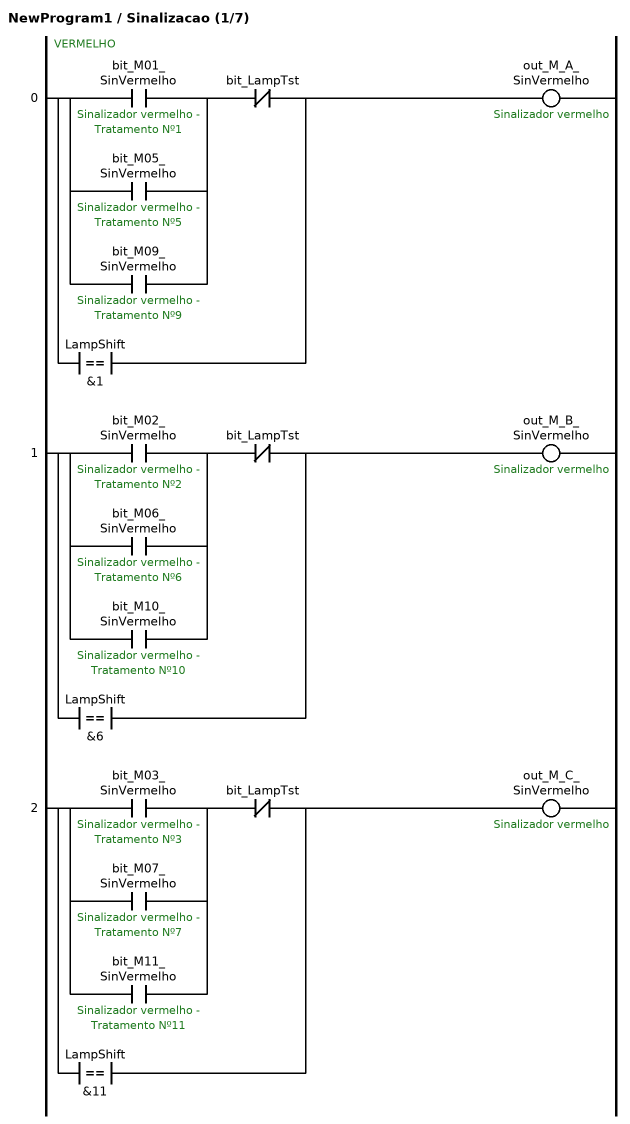
; [picture p48: NewProgram1 / Sinalizacao, rungs 0-2]
; rung 0: VERMELHO
LD bit_M01_SinVermelho  ; Sinalizador vermelho - Tratamento Nº1
OR bit_M05_SinVermelho  ; Sinalizador vermelho - Tratamento Nº5
OR bit_M09_SinVermelho  ; Sinalizador vermelho - Tratamento Nº9
ANDNOT bit_LampTst
OR=(300) LampShift &1
OUT out_M_A_SinVermelho  ; Sinalizador vermelho
; rung 1
LD bit_M02_SinVermelho  ; Sinalizador vermelho - Tratamento Nº2
OR bit_M06_SinVermelho  ; Sinalizador vermelho - Tratamento Nº6
OR bit_M10_SinVermelho  ; Sinalizador vermelho - Tratamento Nº10
ANDNOT bit_LampTst
OR=(300) LampShift &6
OUT out_M_B_SinVermelho  ; Sinalizador vermelho
; rung 2
LD bit_M03_SinVermelho  ; Sinalizador vermelho - Tratamento Nº3
OR bit_M07_SinVermelho  ; Sinalizador vermelho - Tratamento Nº7
OR bit_M11_SinVermelho  ; Sinalizador vermelho - Tratamento Nº11
ANDNOT bit_LampTst
OR=(300) LampShift &11
OUT out_M_C_SinVermelho  ; Sinalizador vermelho

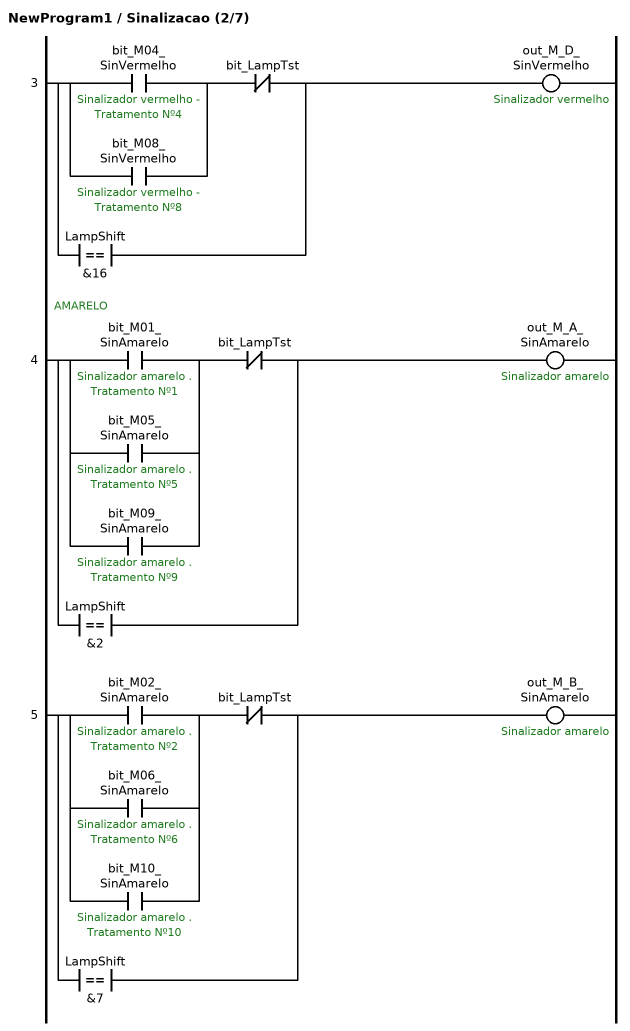
; rung 3
LD bit_M04_SinVermelho  ; Sinalizador vermelho - Tratamento Nº4
OR bit_M08_SinVermelho  ; Sinalizador vermelho - Tratamento Nº8
ANDNOT bit_LampTst
OR=(300) LampShift &16
OUT out_M_D_SinVermelho  ; Sinalizador vermelho
; rung 4: AMARELO
LD bit_M01_SinAmarelo  ; Sinalizador amarelo . Tratamento Nº1
OR bit_M05_SinAmarelo  ; Sinalizador amarelo . Tratamento Nº5
OR bit_M09_SinAmarelo  ; Sinalizador amarelo . Tratamento Nº9
ANDNOT bit_LampTst
OR=(300) LampShift &2
OUT out_M_A_SinAmarelo  ; Sinalizador amarelo
; rung 5
LD bit_M02_SinAmarelo  ; Sinalizador amarelo . Tratamento Nº2
OR bit_M06_SinAmarelo  ; Sinalizador amarelo . Tratamento Nº6
OR bit_M10_SinAmarelo  ; Sinalizador amarelo . Tratamento Nº10
ANDNOT bit_LampTst
OR=(300) LampShift &7
OUT out_M_B_SinAmarelo  ; Sinalizador amarelo

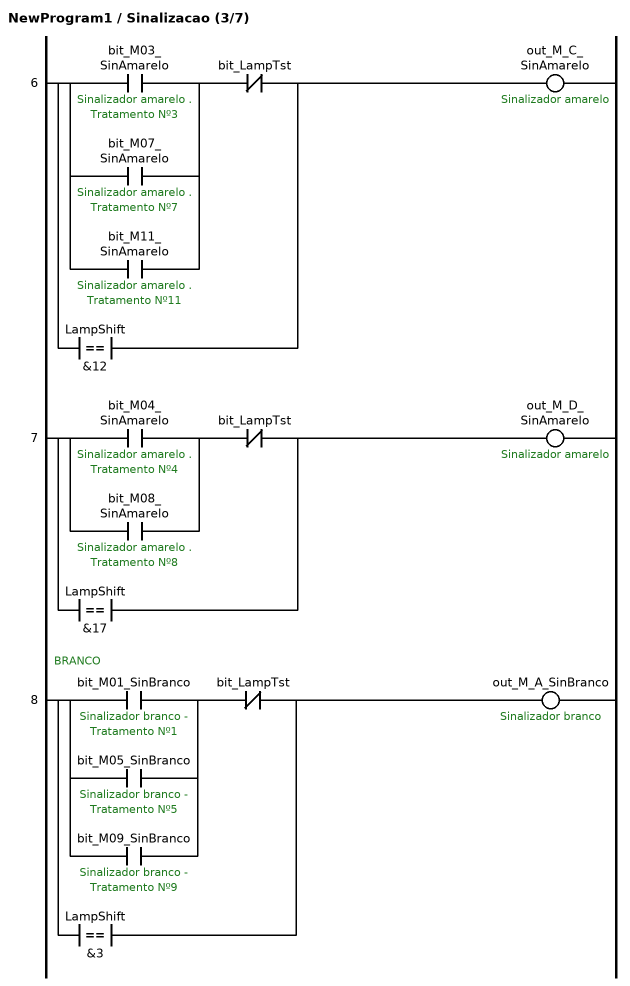
; rung 6
LD bit_M03_SinAmarelo  ; Sinalizador amarelo . Tratamento Nº3
OR bit_M07_SinAmarelo  ; Sinalizador amarelo . Tratamento Nº7
OR bit_M11_SinAmarelo  ; Sinalizador amarelo . Tratamento Nº11
ANDNOT bit_LampTst
OR=(300) LampShift &12
OUT out_M_C_SinAmarelo  ; Sinalizador amarelo
; rung 7
LD bit_M04_SinAmarelo  ; Sinalizador amarelo . Tratamento Nº4
OR bit_M08_SinAmarelo  ; Sinalizador amarelo . Tratamento Nº8
ANDNOT bit_LampTst
OR=(300) LampShift &17
OUT out_M_D_SinAmarelo  ; Sinalizador amarelo
; rung 8: BRANCO
LD bit_M01_SinBranco  ; Sinalizador branco - Tratamento Nº1
OR bit_M05_SinBranco  ; Sinalizador branco - Tratamento Nº5
OR bit_M09_SinBranco  ; Sinalizador branco - Tratamento Nº9
ANDNOT bit_LampTst
OR=(300) LampShift &3
OUT out_M_A_SinBranco  ; Sinalizador branco

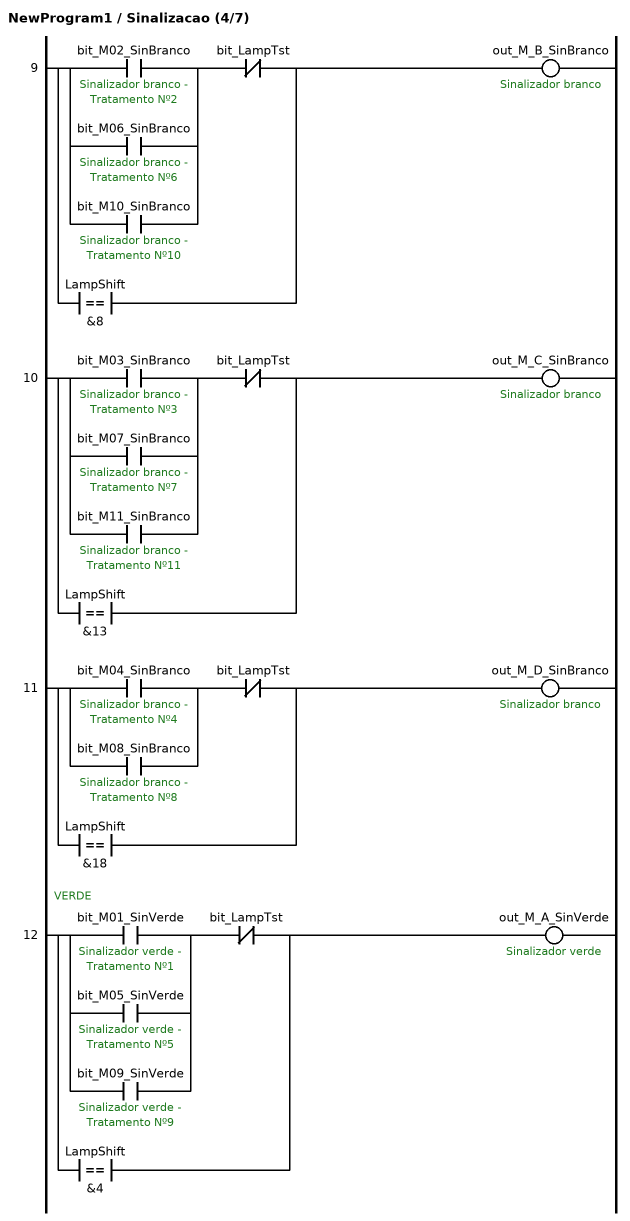
; rung 9
LD bit_M02_SinBranco  ; Sinalizador branco - Tratamento Nº2
OR bit_M06_SinBranco  ; Sinalizador branco - Tratamento Nº6
OR bit_M10_SinBranco  ; Sinalizador branco - Tratamento Nº10
ANDNOT bit_LampTst
OR=(300) LampShift &8
OUT out_M_B_SinBranco  ; Sinalizador branco
; rung 10
LD bit_M03_SinBranco  ; Sinalizador branco - Tratamento Nº3
OR bit_M07_SinBranco  ; Sinalizador branco - Tratamento Nº7
OR bit_M11_SinBranco  ; Sinalizador branco - Tratamento Nº11
ANDNOT bit_LampTst
OR=(300) LampShift &13
OUT out_M_C_SinBranco  ; Sinalizador branco
; rung 11
LD bit_M04_SinBranco  ; Sinalizador branco - Tratamento Nº4
OR bit_M08_SinBranco  ; Sinalizador branco - Tratamento Nº8
ANDNOT bit_LampTst
OR=(300) LampShift &18
OUT out_M_D_SinBranco  ; Sinalizador branco
; rung 12: VERDE
LD bit_M01_SinVerde  ; Sinalizador verde - Tratamento Nº1
OR bit_M05_SinVerde  ; Sinalizador verde - Tratamento Nº5
OR bit_M09_SinVerde  ; Sinalizador verde - Tratamento Nº9
ANDNOT bit_LampTst
OR=(300) LampShift &4
OUT out_M_A_SinVerde  ; Sinalizador verde

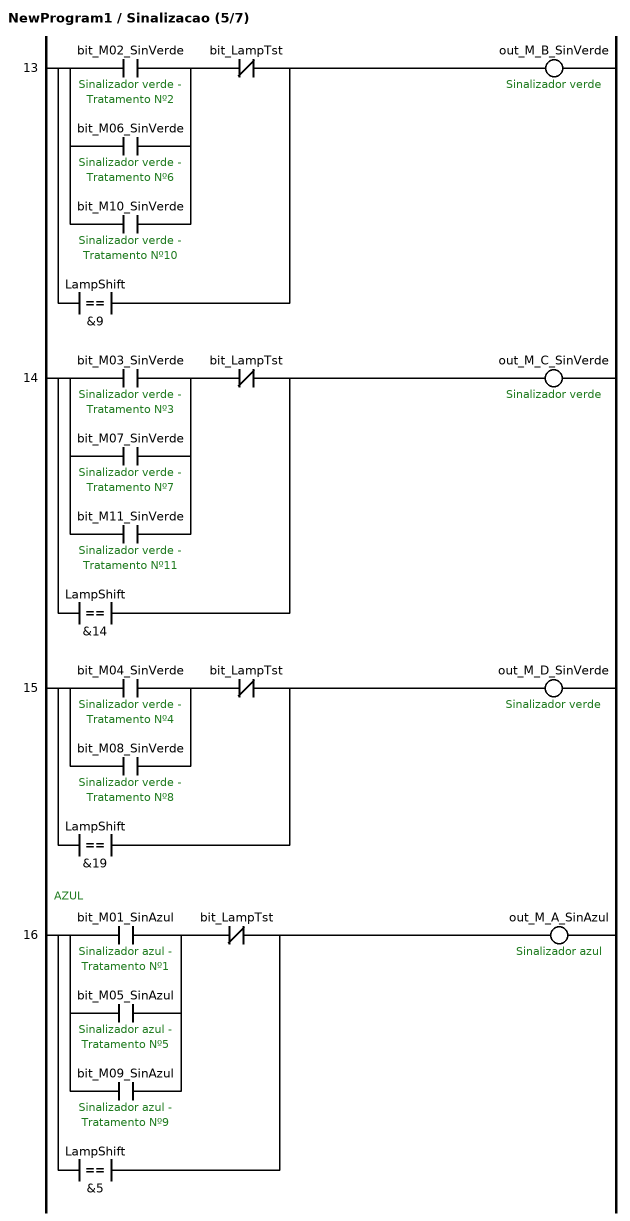
; rung 13
LD bit_M02_SinVerde  ; Sinalizador verde - Tratamento Nº2
OR bit_M06_SinVerde  ; Sinalizador verde - Tratamento Nº6
OR bit_M10_SinVerde  ; Sinalizador verde - Tratamento Nº10
ANDNOT bit_LampTst
OR=(300) LampShift &9
OUT out_M_B_SinVerde  ; Sinalizador verde
; rung 14
LD bit_M03_SinVerde  ; Sinalizador verde - Tratamento Nº3
OR bit_M07_SinVerde  ; Sinalizador verde - Tratamento Nº7
OR bit_M11_SinVerde  ; Sinalizador verde - Tratamento Nº11
ANDNOT bit_LampTst
OR=(300) LampShift &14
OUT out_M_C_SinVerde  ; Sinalizador verde
; rung 15
LD bit_M04_SinVerde  ; Sinalizador verde - Tratamento Nº4
OR bit_M08_SinVerde  ; Sinalizador verde - Tratamento Nº8
ANDNOT bit_LampTst
OR=(300) LampShift &19
OUT out_M_D_SinVerde  ; Sinalizador verde
; rung 16: AZUL
LD bit_M01_SinAzul  ; Sinalizador azul - Tratamento Nº1
OR bit_M05_SinAzul  ; Sinalizador azul - Tratamento Nº5
OR bit_M09_SinAzul  ; Sinalizador azul - Tratamento Nº9
ANDNOT bit_LampTst
OR=(300) LampShift &5
OUT out_M_A_SinAzul  ; Sinalizador azul

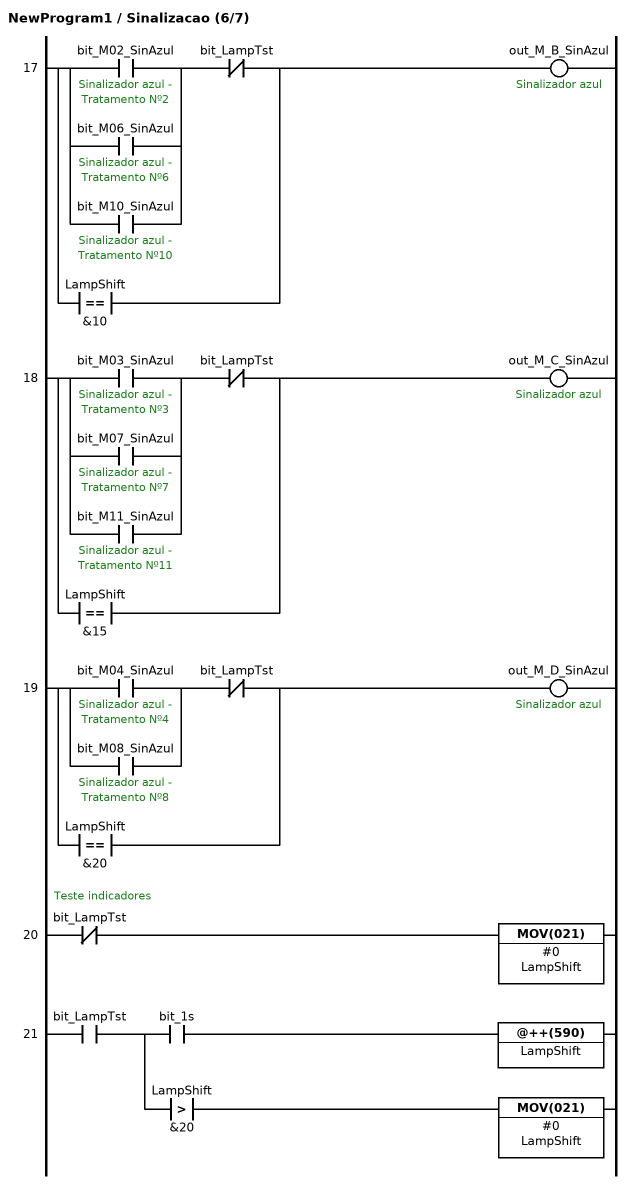
; rung 17
LD bit_M02_SinAzul  ; Sinalizador azul - Tratamento Nº2
OR bit_M06_SinAzul  ; Sinalizador azul - Tratamento Nº6
OR bit_M10_SinAzul  ; Sinalizador azul - Tratamento Nº10
ANDNOT bit_LampTst
OR=(300) LampShift &10
OUT out_M_B_SinAzul  ; Sinalizador azul
; rung 18
LD bit_M03_SinAzul  ; Sinalizador azul - Tratamento Nº3
OR bit_M07_SinAzul  ; Sinalizador azul - Tratamento Nº7
OR bit_M11_SinAzul  ; Sinalizador azul - Tratamento Nº11
ANDNOT bit_LampTst
OR=(300) LampShift &15
OUT out_M_C_SinAzul  ; Sinalizador azul
; rung 19
LD bit_M04_SinAzul  ; Sinalizador azul - Tratamento Nº4
OR bit_M08_SinAzul  ; Sinalizador azul - Tratamento Nº8
ANDNOT bit_LampTst
OR=(300) LampShift &20
OUT out_M_D_SinAzul  ; Sinalizador azul
; rung 20: Teste indicadores
LDNOT bit_LampTst
MOV(021) #0 LampShift
; rung 21
LD bit_LampTst
OUT TR0
AND bit_1s
@++(590) LampShift
LD TR0
AND>(320) LampShift &20
MOV(021) #0 LampShift

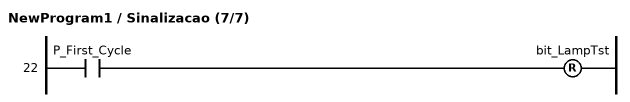
; rung 22
LD P_First_Cycle
RSET bit_LampTst

### Section RqstForTransfer

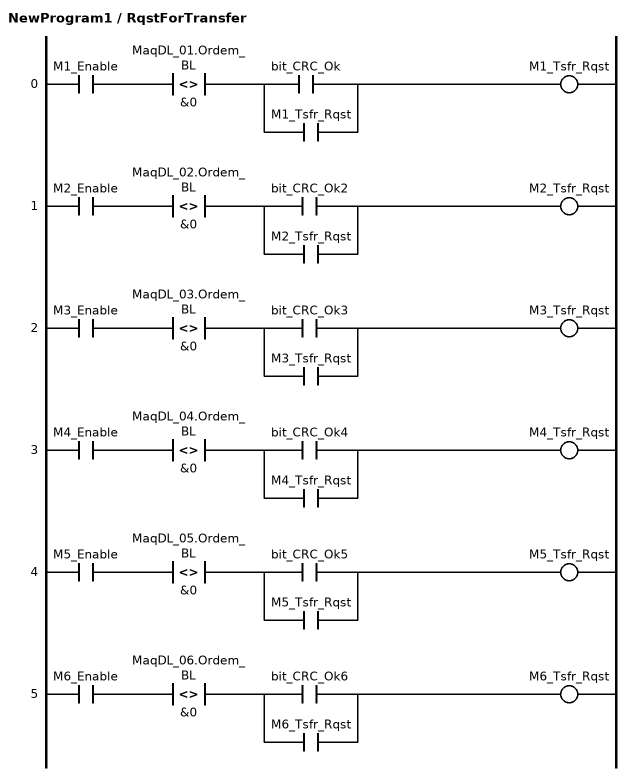
; rung 0
LD M1_Enable
AND<>(305) MaqDL_01.Ordem_BL &0
LD bit_CRC_Ok
OR M1_Tsfr_Rqst
ANDLD
OUT M1_Tsfr_Rqst
; rung 1
LD M2_Enable
AND<>(305) MaqDL_02.Ordem_BL &0
LD bit_CRC_Ok2
OR M2_Tsfr_Rqst
ANDLD
OUT M2_Tsfr_Rqst
; rung 2
LD M3_Enable
AND<>(305) MaqDL_03.Ordem_BL &0
LD bit_CRC_Ok3
OR M3_Tsfr_Rqst
ANDLD
OUT M3_Tsfr_Rqst
; rung 3
LD M4_Enable
AND<>(305) MaqDL_04.Ordem_BL &0
LD bit_CRC_Ok4
OR M4_Tsfr_Rqst
ANDLD
OUT M4_Tsfr_Rqst
; rung 4
LD M5_Enable
AND<>(305) MaqDL_05.Ordem_BL &0
LD bit_CRC_Ok5
OR M5_Tsfr_Rqst
ANDLD
OUT M5_Tsfr_Rqst
; rung 5
LD M6_Enable
AND<>(305) MaqDL_06.Ordem_BL &0
LD bit_CRC_Ok6
OR M6_Tsfr_Rqst
ANDLD
OUT M6_Tsfr_Rqst

### Section END

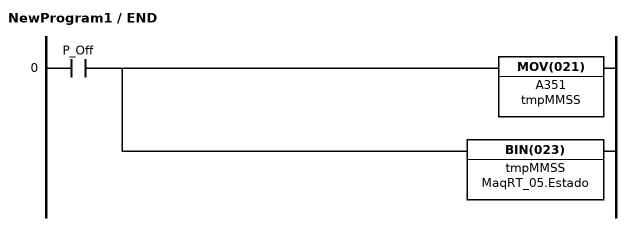
; rung 0
LD P_Off
MOV(021) A351 tmpMMSS
BIN(023) tmpMMSS MaqRT_05.Estado
; rung 1
END(001)

## Function block _CPU010_SendData (Omron library block, body left out)

## Function block ARRAY_COPY
VAR_INPUT
  NPos : INT;
END_VAR
VAR_IN_OUT
  ArIN : ARRAY[0..0] OF WORD;
  ArOUT : ARRAY[0..49] OF WORD;
END_VAR
VAR
  i : INT;
END_VAR
FOR i:= 0 TO 49 DO 
	ArOUT [i]:= 0;
END_FOR; 
FOR i:= 0 TO (NPos -1) DO 
	ArOUT [i]:= ArIN [i];
END_FOR; 

## Function block CopyRcp
VAR_INPUT
  Start : BOOL;
END_VAR
VAR_IN_OUT
  Dados : MqDL;
END_VAR
IF Start THEN
Dados.Cliente[0]:= Dados.Cliente_BL[0];
Dados.Cliente[1]:= Dados.Cliente_BL[1];
Dados.Cliente[2]:= Dados.Cliente_BL[2];
Dados.Cliente[3]:= Dados.Cliente_BL[3];
Dados.Cliente[4]:= Dados.Cliente_BL[4];
Dados.Cliente[5]:= Dados.Cliente_BL[5];
Dados.Cliente[6]:= Dados.Cliente_BL[6];
Dados.Cliente[7]:= Dados.Cliente_BL[7];
Dados.Cliente[8]:= Dados.Cliente_BL[8];
Dados.Cliente[9]:= Dados.Cliente_BL[9];
Dados.Cliente[10]:= Dados.Cliente_BL[10];
Dados.Cliente[11]:= Dados.Cliente_BL[11];
Dados.Cliente[12]:= Dados.Cliente_BL[12];
Dados.Cliente[13]:= Dados.Cliente_BL[13];
Dados.Cliente[14]:= Dados.Cliente_BL[14];
Dados.Cliente[15]:= Dados.Cliente_BL[15];
Dados.Cliente[16]:= Dados.Cliente_BL[16];
Dados.Cliente[17]:= Dados.Cliente_BL[17];
Dados.Cliente[18]:= Dados.Cliente_BL[18];
Dados.Cliente[19]:= Dados.Cliente_BL[19];
Dados.Cliente[20]:= Dados.Cliente_BL[20];
Dados.Cliente[21]:= Dados.Cliente_BL[21];
Dados.Cliente[22]:= Dados.Cliente_BL[22];
Dados.Cliente[23]:= Dados.Cliente_BL[23];
Dados.Cliente[24]:= Dados.Cliente_BL[24];
Dados.Cliente[25]:= Dados.Cliente_BL[25];
Dados.Cliente[26]:= Dados.Cliente_BL[26];
Dados.Cliente[27]:= Dados.Cliente_BL[27];
Dados.Cliente[28]:= Dados.Cliente_BL[28];
Dados.Cliente[29]:= Dados.Cliente_BL[29];
Dados.Cliente[30]:= Dados.Cliente_BL[30];
Dados.Cliente[31]:= Dados.Cliente_BL[31];
Dados.Cliente[32]:= Dados.Cliente_BL[32];
Dados.Cliente[33]:= Dados.Cliente_BL[33];
Dados.Cliente[34]:= Dados.Cliente_BL[34];
Dados.Cliente[35]:= Dados.Cliente_BL[35];
Dados.Cliente[36]:= Dados.Cliente_BL[36];
Dados.Cliente[37]:= Dados.Cliente_BL[37];
Dados.Cliente[38]:= Dados.Cliente_BL[38];
Dados.Cliente[39]:= Dados.Cliente_BL[39];
Dados.Cliente[40]:= Dados.Cliente_BL[40];
Dados.Cliente[41]:= Dados.Cliente_BL[41];
Dados.Cliente[42]:= Dados.Cliente_BL[42];
Dados.Cliente[43]:= Dados.Cliente_BL[43];
Dados.Cliente[44]:= Dados.Cliente_BL[44];
Dados.Cliente[45]:= Dados.Cliente_BL[45];
Dados.Cliente[46]:= Dados.Cliente_BL[46];
Dados.Cliente[47]:= Dados.Cliente_BL[47];
Dados.Cliente[48]:= Dados.Cliente_BL[48];
Dados.Cliente[49]:= Dados.Cliente_BL[49];

Dados.Artigo[0]:= Dados.Artigo_BL[0];
Dados.Artigo[1]:= Dados.Artigo_BL[1];
Dados.Artigo[2]:= Dados.Artigo_BL[2];
Dados.Artigo[3]:= Dados.Artigo_BL[3];
Dados.Artigo[4]:= Dados.Artigo_BL[4];
Dados.Artigo[5]:= Dados.Artigo_BL[5];
Dados.Artigo[6]:= Dados.Artigo_BL[6];
Dados.Artigo[7]:= Dados.Artigo_BL[7];
Dados.Artigo[8]:= Dados.Artigo_BL[8];
Dados.Artigo[9]:= Dados.Artigo_BL[9];
Dados.Artigo[10]:= Dados.Artigo_BL[10];
Dados.Artigo[11]:= Dados.Artigo_BL[11];
Dados.Artigo[12]:= Dados.Artigo_BL[12];
Dados.Artigo[13]:= Dados.Artigo_BL[13];
Dados.Artigo[14]:= Dados.Artigo_BL[14];
Dados.Artigo[15]:= Dados.Artigo_BL[15];
Dados.Artigo[16]:= Dados.Artigo_BL[16];
Dados.Artigo[17]:= Dados.Artigo_BL[17];
Dados.Artigo[18]:= Dados.Artigo_BL[18];
Dados.Artigo[19]:= Dados.Artigo_BL[19];
Dados.Artigo[20]:= Dados.Artigo_BL[20];
Dados.Artigo[21]:= Dados.Artigo_BL[21];
Dados.Artigo[22]:= Dados.Artigo_BL[22];
Dados.Artigo[23]:= Dados.Artigo_BL[23];
Dados.Artigo[24]:= Dados.Artigo_BL[24];
Dados.Artigo[25]:= Dados.Artigo_BL[25];
Dados.Artigo[26]:= Dados.Artigo_BL[26];
Dados.Artigo[27]:= Dados.Artigo_BL[27];
Dados.Artigo[28]:= Dados.Artigo_BL[28];
Dados.Artigo[29]:= Dados.Artigo_BL[29];
Dados.Artigo[30]:= Dados.Artigo_BL[30];
Dados.Artigo[31]:= Dados.Artigo_BL[31];
Dados.Artigo[32]:= Dados.Artigo_BL[32];
Dados.Artigo[33]:= Dados.Artigo_BL[33];
Dados.Artigo[34]:= Dados.Artigo_BL[34];
Dados.Artigo[35]:= Dados.Artigo_BL[35];
Dados.Artigo[36]:= Dados.Artigo_BL[36];
Dados.Artigo[37]:= Dados.Artigo_BL[37];
Dados.Artigo[38]:= Dados.Artigo_BL[38];
Dados.Artigo[39]:= Dados.Artigo_BL[39];
Dados.Artigo[40]:= Dados.Artigo_BL[40];
Dados.Artigo[41]:= Dados.Artigo_BL[41];
Dados.Artigo[42]:= Dados.Artigo_BL[42];
Dados.Artigo[43]:= Dados.Artigo_BL[43];
Dados.Artigo[44]:= Dados.Artigo_BL[44];
Dados.Artigo[45]:= Dados.Artigo_BL[45];
Dados.Artigo[46]:= Dados.Artigo_BL[46];
Dados.Artigo[47]:= Dados.Artigo_BL[47];
Dados.Artigo[48]:= Dados.Artigo_BL[48];
Dados.Artigo[49]:= Dados.Artigo_BL[49];

Dados.Encomenda[0]:= Dados.Encomenda_BL[0];
Dados.Encomenda[1]:= Dados.Encomenda_BL[1];
Dados.Encomenda[2]:= Dados.Encomenda_BL[2];
Dados.Encomenda[3]:= Dados.Encomenda_BL[3];
Dados.Encomenda[4]:= Dados.Encomenda_BL[4];
Dados.Encomenda[5]:= Dados.Encomenda_BL[5];
Dados.Encomenda[6]:= Dados.Encomenda_BL[6];
Dados.Encomenda[7]:= Dados.Encomenda_BL[7];
Dados.Encomenda[8]:= Dados.Encomenda_BL[8];
Dados.Encomenda[9]:= Dados.Encomenda_BL[9];
Dados.Encomenda[10]:= Dados.Encomenda_BL[10];
Dados.Encomenda[11]:= Dados.Encomenda_BL[11];
Dados.Encomenda[12]:= Dados.Encomenda_BL[12];
Dados.Encomenda[13]:= Dados.Encomenda_BL[13];
Dados.Encomenda[14]:= Dados.Encomenda_BL[14];
Dados.Encomenda[15]:= Dados.Encomenda_BL[15];
Dados.Encomenda[16]:= Dados.Encomenda_BL[16];
Dados.Encomenda[17]:= Dados.Encomenda_BL[17];
Dados.Encomenda[18]:= Dados.Encomenda_BL[18];
Dados.Encomenda[19]:= Dados.Encomenda_BL[19];
Dados.Encomenda[20]:= Dados.Encomenda_BL[20];
Dados.Encomenda[21]:= Dados.Encomenda_BL[21];
Dados.Encomenda[22]:= Dados.Encomenda_BL[22];
Dados.Encomenda[23]:= Dados.Encomenda_BL[23];
Dados.Encomenda[24]:= Dados.Encomenda_BL[24];
Dados.Encomenda[25]:= Dados.Encomenda_BL[25];
Dados.Encomenda[26]:= Dados.Encomenda_BL[26];
Dados.Encomenda[27]:= Dados.Encomenda_BL[27];
Dados.Encomenda[28]:= Dados.Encomenda_BL[28];
Dados.Encomenda[29]:= Dados.Encomenda_BL[29];
Dados.Encomenda[30]:= Dados.Encomenda_BL[30];
Dados.Encomenda[31]:= Dados.Encomenda_BL[31];
Dados.Encomenda[32]:= Dados.Encomenda_BL[32];
Dados.Encomenda[33]:= Dados.Encomenda_BL[33];
Dados.Encomenda[34]:= Dados.Encomenda_BL[34];
Dados.Encomenda[35]:= Dados.Encomenda_BL[35];
Dados.Encomenda[36]:= Dados.Encomenda_BL[36];
Dados.Encomenda[37]:= Dados.Encomenda_BL[37];
Dados.Encomenda[38]:= Dados.Encomenda_BL[38];
Dados.Encomenda[39]:= Dados.Encomenda_BL[39];
Dados.Encomenda[40]:= Dados.Encomenda_BL[40];
Dados.Encomenda[41]:= Dados.Encomenda_BL[41];
Dados.Encomenda[42]:= Dados.Encomenda_BL[42];
Dados.Encomenda[43]:= Dados.Encomenda_BL[43];
Dados.Encomenda[44]:= Dados.Encomenda_BL[44];
Dados.Encomenda[45]:= Dados.Encomenda_BL[45];
Dados.Encomenda[46]:= Dados.Encomenda_BL[46];
Dados.Encomenda[47]:= Dados.Encomenda_BL[47];
Dados.Encomenda[48]:= Dados.Encomenda_BL[48];
Dados.Encomenda[49]:= Dados.Encomenda_BL[49];

Dados.NomeReceita[0]:= Dados.NomeReceita_BL[0];
Dados.NomeReceita[1]:= Dados.NomeReceita_BL[1];
Dados.NomeReceita[2]:= Dados.NomeReceita_BL[2];
Dados.NomeReceita[3]:= Dados.NomeReceita_BL[3];
Dados.NomeReceita[4]:= Dados.NomeReceita_BL[4];
Dados.NomeReceita[5]:= Dados.NomeReceita_BL[5];
Dados.NomeReceita[6]:= Dados.NomeReceita_BL[6];
Dados.NomeReceita[7]:= Dados.NomeReceita_BL[7];
Dados.NomeReceita[8]:= Dados.NomeReceita_BL[8];
Dados.NomeReceita[9]:= Dados.NomeReceita_BL[9];
Dados.NomeReceita[10]:= Dados.NomeReceita_BL[10];
Dados.NomeReceita[11]:= Dados.NomeReceita_BL[11];
Dados.NomeReceita[12]:= Dados.NomeReceita_BL[12];
Dados.NomeReceita[13]:= Dados.NomeReceita_BL[13];
Dados.NomeReceita[14]:= Dados.NomeReceita_BL[14];
Dados.NomeReceita[15]:= Dados.NomeReceita_BL[15];
Dados.NomeReceita[16]:= Dados.NomeReceita_BL[16];
Dados.NomeReceita[17]:= Dados.NomeReceita_BL[17];
Dados.NomeReceita[18]:= Dados.NomeReceita_BL[18];
Dados.NomeReceita[19]:= Dados.NomeReceita_BL[19];
Dados.NomeReceita[20]:= Dados.NomeReceita_BL[20];
Dados.NomeReceita[21]:= Dados.NomeReceita_BL[21];
Dados.NomeReceita[22]:= Dados.NomeReceita_BL[22];
Dados.NomeReceita[23]:= Dados.NomeReceita_BL[23];
Dados.NomeReceita[24]:= Dados.NomeReceita_BL[24];
Dados.NomeReceita[25]:= Dados.NomeReceita_BL[25];
Dados.NomeReceita[26]:= Dados.NomeReceita_BL[26];
Dados.NomeReceita[27]:= Dados.NomeReceita_BL[27];
Dados.NomeReceita[28]:= Dados.NomeReceita_BL[28];
Dados.NomeReceita[29]:= Dados.NomeReceita_BL[29];
Dados.NomeReceita[30]:= Dados.NomeReceita_BL[30];
Dados.NomeReceita[31]:= Dados.NomeReceita_BL[31];
Dados.NomeReceita[32]:= Dados.NomeReceita_BL[32];
Dados.NomeReceita[33]:= Dados.NomeReceita_BL[33];
Dados.NomeReceita[34]:= Dados.NomeReceita_BL[34];
Dados.NomeReceita[35]:= Dados.NomeReceita_BL[35];
Dados.NomeReceita[36]:= Dados.NomeReceita_BL[36];
Dados.NomeReceita[37]:= Dados.NomeReceita_BL[37];
Dados.NomeReceita[38]:= Dados.NomeReceita_BL[38];
Dados.NomeReceita[39]:= Dados.NomeReceita_BL[39];
Dados.NomeReceita[40]:= Dados.NomeReceita_BL[40];
Dados.NomeReceita[41]:= Dados.NomeReceita_BL[41];
Dados.NomeReceita[42]:= Dados.NomeReceita_BL[42];
Dados.NomeReceita[43]:= Dados.NomeReceita_BL[43];
Dados.NomeReceita[44]:= Dados.NomeReceita_BL[44];
Dados.NomeReceita[45]:= Dados.NomeReceita_BL[45];
Dados.NomeReceita[46]:= Dados.NomeReceita_BL[46];
Dados.NomeReceita[47]:= Dados.NomeReceita_BL[47];
Dados.NomeReceita[48]:= Dados.NomeReceita_BL[48];
Dados.NomeReceita[49]:= Dados.NomeReceita_BL[49];

Dados.DataExpedic[0]:= Dados.DataExpedic_BL[0];
Dados.DataExpedic[1]:= Dados.DataExpedic_BL[1];
Dados.DataExpedic[2]:= Dados.DataExpedic_BL[2];
Dados.DataExpedic[3]:= Dados.DataExpedic_BL[3];

Dados.QtdEncom:= Dados.QtdEncom_BL;
Dados.QtdReal:= Dados.QtdReal_BL;

END_IF;

## Function block CopySteps
VAR_OUTPUT
  Rcp_Ok : BOOL;
END_VAR
VAR_IN_OUT
  Recipe : s_of;
  Steps : ARRAY[0..11] OF Passos;
END_VAR
Steps[0].f:= Recipe.prg.pss[0].f;
Steps[0].p1:= Recipe.prg.pss[0].p1;
Steps[0].p2:= Recipe.prg.pss[0].p2 ;

Steps[1].f:= Recipe.prg.pss[1].f;
Steps[1].p1:= Recipe.prg.pss[1].p1;
Steps[1].p2:= Recipe.prg.pss[1].p2 ;

Steps[2].f:= Recipe.prg.pss[2].f;
Steps[2].p1:= Recipe.prg.pss[2].p1;
Steps[2].p2:= Recipe.prg.pss[2].p2 ;

Steps[3].f:= Recipe.prg.pss[3].f;
Steps[3].p1:= Recipe.prg.pss[3].p1;
Steps[3].p2:= Recipe.prg.pss[3].p2 ;

Steps[4].f:= Recipe.prg.pss[4].f;
Steps[4].p1:= Recipe.prg.pss[4].p1;
Steps[4].p2:= Recipe.prg.pss[4].p2 ;

Steps[5].f:= Recipe.prg.pss[5].f;
Steps[5].p1:= Recipe.prg.pss[5].p1;
Steps[5].p2:= Recipe.prg.pss[5].p2 ;

Steps[6].f:= Recipe.prg.pss[6].f;
Steps[6].p1:= Recipe.prg.pss[6].p1;
Steps[6].p2:= Recipe.prg.pss[6].p2 ;

Steps[7].f:= Recipe.prg.pss[7].f;
Steps[7].p1:= Recipe.prg.pss[7].p1;
Steps[7].p2:= Recipe.prg.pss[7].p2 ;

Steps[8].f:= Recipe.prg.pss[8].f;
Steps[8].p1:= Recipe.prg.pss[8].p1;
Steps[8].p2:= Recipe.prg.pss[8].p2 ;

Steps[9].f:= Recipe.prg.pss[9].f;
Steps[9].p1:= Recipe.prg.pss[9].p1;
Steps[9].p2:= Recipe.prg.pss[9].p2 ;

Steps[10].f:= Recipe.prg.pss[10].f;
Steps[10].p1:= Recipe.prg.pss[10].p1;
Steps[10].p2:= Recipe.prg.pss[10].p2 ;

Steps[11].f:= Recipe.prg.pss[11].f;
Steps[11].p1:= Recipe.prg.pss[11].p1;
Steps[11].p2:= Recipe.prg.pss[11].p2 ;

Rcp_Ok:= TRUE;

## Function block CRC16
VAR_INPUT
  Bytes_Qty : INT;
  Swap : BOOL;  (* Swap LSB with MSB *)
  CRC_Ini : WORD;
END_VAR
VAR_OUTPUT
  CRC16 : WORD;
END_VAR
VAR_IN_OUT
  Str : STRING;
END_VAR
VAR
  Flip_Flop : BOOL;
  Next_Byte : WORD;
  CRC_Temp : WORD;
  i : INT;
  aux_Byte : WORD;
END_VAR

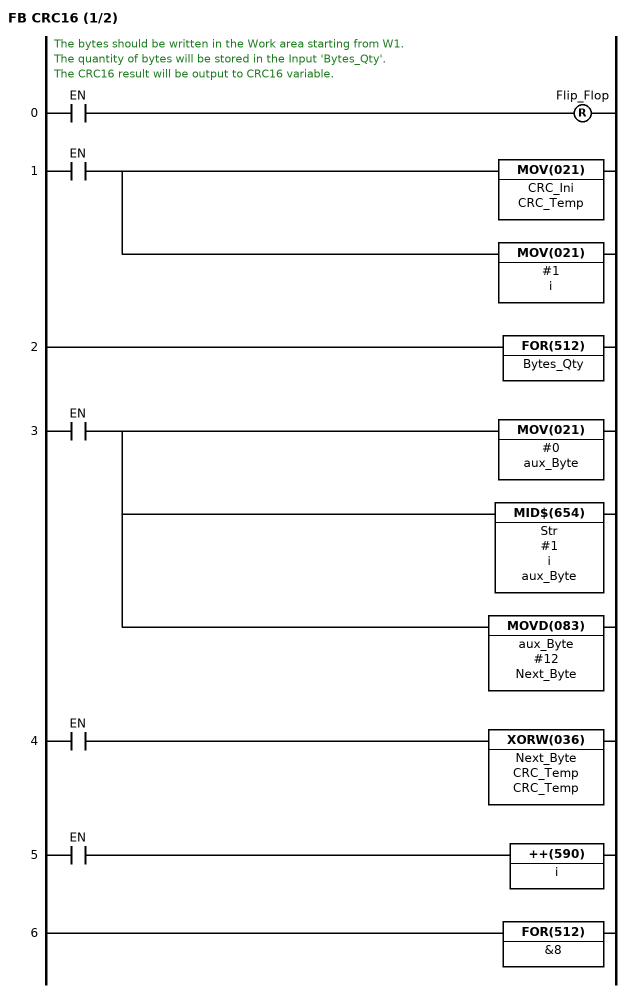
; rung 0: The bytes should be written in the Work area starting from W1. / The quantity of bytes will be stored in the Input 'Bytes_Qty'. / The CRC16 result will be output to CRC16 variable.
LD EN
RSET Flip_Flop
; rung 1
LD EN
MOV(021) CRC_Ini CRC_Temp
MOV(021) #1 i
; rung 2
FOR(512) Bytes_Qty
; rung 3
LD EN
MOV(021) #0 aux_Byte
MID$(654) Str #1 i aux_Byte
MOVD(083) aux_Byte #12 Next_Byte
; rung 4
LD EN
XORW(036) Next_Byte CRC_Temp CRC_Temp
; rung 5
LD EN
++(590) i
; rung 6
FOR(512) &8

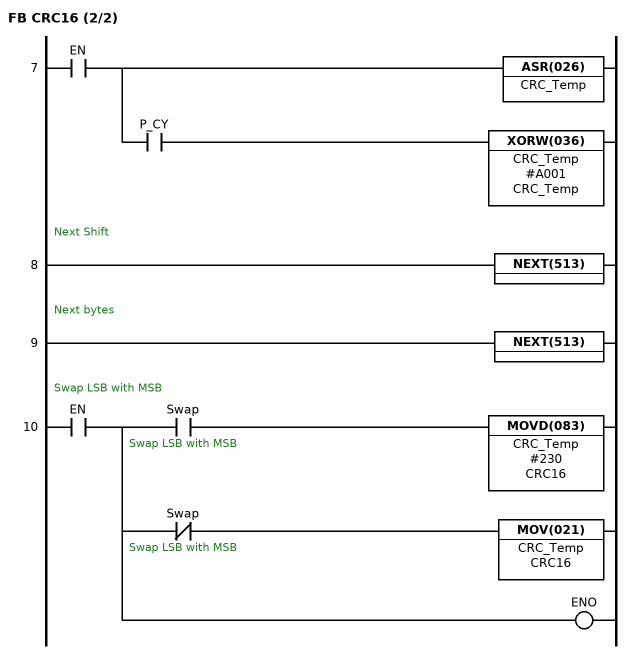
; rung 7
LD EN
ASR(026) CRC_Temp
AND P_CY
XORW(036) CRC_Temp #A001 CRC_Temp
; rung 8: Next Shift
NEXT(513)
; rung 9: Next bytes
NEXT(513)
; rung 10: Swap LSB with MSB
LD EN
OUT TR0
AND Swap  ; Swap LSB with MSB
MOVD(083) CRC_Temp #230 CRC16
LD TR0
ANDNOT Swap  ; Swap LSB with MSB
MOV(021) CRC_Temp CRC16
LD TR0
OUT ENO

## Function block DWord_To_Real
VAR_INPUT
  A : DWORD;
END_VAR
VAR_OUTPUT
  B : REAL;
END_VAR
VAR
  c : DINT;
END_VAR
c:= DWORD_TO_DINT(A);
B:= DINT_TO_REAL(c);

## Function block Empty_LSP
VAR_INPUT
  Fst_indx : INT;
  Lst_indx : INT;
END_VAR
VAR_OUTPUT
  Empty_Pos : INT;
  Last_Position : BOOL;
END_VAR
VAR_IN_OUT
  Ary : ARRAY[0..99] OF INT;
END_VAR
VAR
  itr : INT;
  Loop_Stop : BOOL;
END_VAR
Loop_Stop := FALSE;

FOR itr := Fst_indx TO Lst_indx DO
IF Ary[itr]=0 AND  NOT Loop_Stop THEN
	Empty_Pos := itr;
	Loop_Stop := TRUE;
END_IF;
END_FOR;

IF Ary[Lst_indx] <> 0 THEN
	Last_Position := TRUE;
	Empty_Pos := -1;
ELSE
	Last_Position := FALSE;
END_IF;

## Function block FIFO
; This function finds the least significant position of a arry. / The seeking area can be limited by firsr arry (FstAry) and last Array (LstAry) which are the inputs of function block.
VAR_INPUT
  Line_Free : BOOL;
  cmd_EN : BOOL;
  M1_Rqst : BOOL;
  M2_Rqst : BOOL;
  M3_Rqst : BOOL;
  M4_Rqst : BOOL;
  M5_Rqst : BOOL;
  M6_Rqst : BOOL;
  Table_Length : INT;
END_VAR
VAR_OUTPUT
  Actv_M : INT;
  cmd_M1 : BOOL;
  cmd_M2 : BOOL;
  cmd_M3 : BOOL;
  cmd_M4 : BOOL;
  cmd_M5 : BOOL;
  cmd_M6 : BOOL;
  Table_Full : BOOL;
END_VAR
VAR_IN_OUT
  Table : ARRAY[0..99] OF INT;
END_VAR
VAR
  M_Rqst_tmp : INT;
  Empty_in_Table : Empty_LSP;
  Empty_Position : INT;
  Shift_Table : Shift_Ary;
  cmd_Shift : BOOL;
  Tabel_LstIndx : INT;
END_VAR

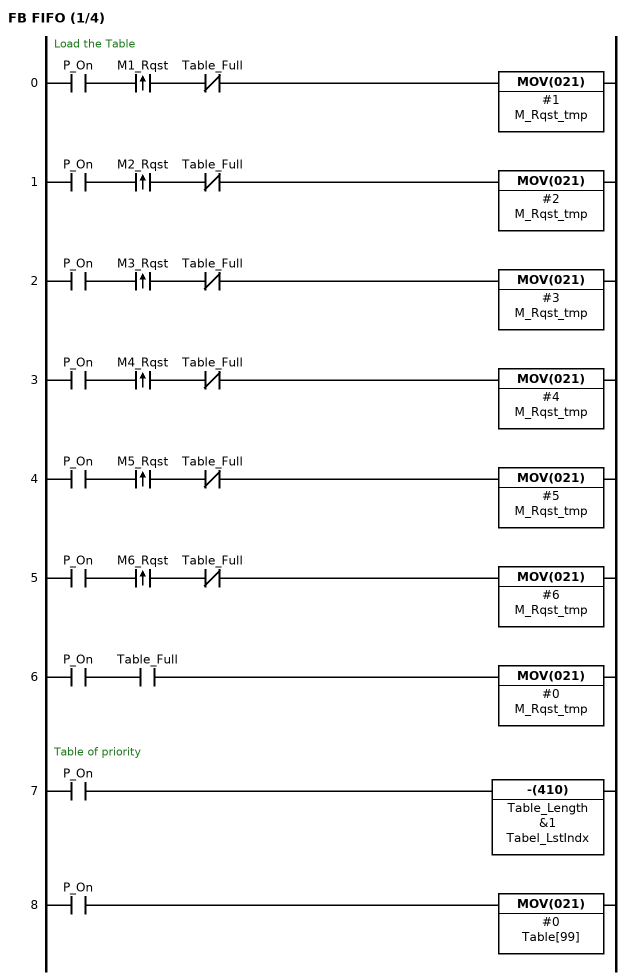
; rung 0: Load the Table
LD P_On
@AND M1_Rqst
ANDNOT Table_Full
MOV(021) #1 M_Rqst_tmp
; rung 1
LD P_On
@AND M2_Rqst
ANDNOT Table_Full
MOV(021) #2 M_Rqst_tmp
; rung 2
LD P_On
@AND M3_Rqst
ANDNOT Table_Full
MOV(021) #3 M_Rqst_tmp
; rung 3
LD P_On
@AND M4_Rqst
ANDNOT Table_Full
MOV(021) #4 M_Rqst_tmp
; rung 4
LD P_On
@AND M5_Rqst
ANDNOT Table_Full
MOV(021) #5 M_Rqst_tmp
; rung 5
LD P_On
@AND M6_Rqst
ANDNOT Table_Full
MOV(021) #6 M_Rqst_tmp
; rung 6
LD P_On
AND Table_Full
MOV(021) #0 M_Rqst_tmp
; rung 7: Table of priority
LD P_On
-(410) Table_Length &1 Tabel_LstIndx
; rung 8
LD P_On
MOV(021) #0 Table[99]

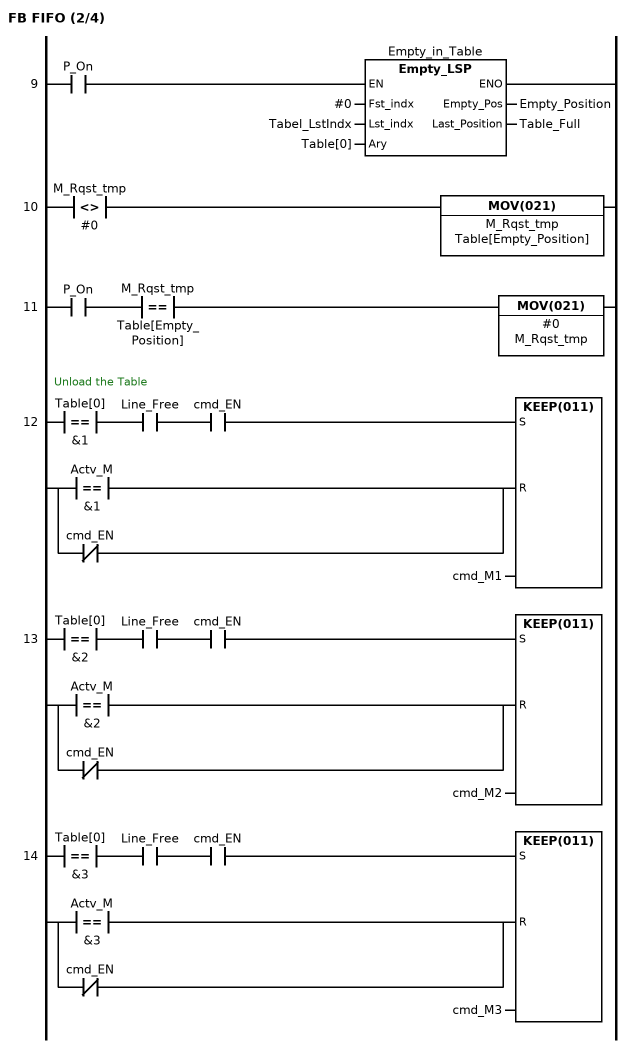
; rung 9
LD P_On
CALL Empty_in_Table : Empty_LSP (Fst_indx := #0, Lst_indx := Tabel_LstIndx, Ary := Table[0], Empty_Pos => Empty_Position, Last_Position => Table_Full)
; rung 10
LD<>(305) M_Rqst_tmp #0
MOV(021) M_Rqst_tmp Table[Empty_Position]
; rung 11
LD P_On
AND=(300) M_Rqst_tmp Table[Empty_Position]
MOV(021) #0 M_Rqst_tmp
; rung 12: Unload the Table
LD=(300) Table[0] &1
AND Line_Free
AND cmd_EN
LD=(300) Actv_M &1
ORNOT cmd_EN
KEEP(011) cmd_M1
; rung 13
LD=(300) Table[0] &2
AND Line_Free
AND cmd_EN
LD=(300) Actv_M &2
ORNOT cmd_EN
KEEP(011) cmd_M2
; rung 14
LD=(300) Table[0] &3
AND Line_Free
AND cmd_EN
LD=(300) Actv_M &3
ORNOT cmd_EN
KEEP(011) cmd_M3

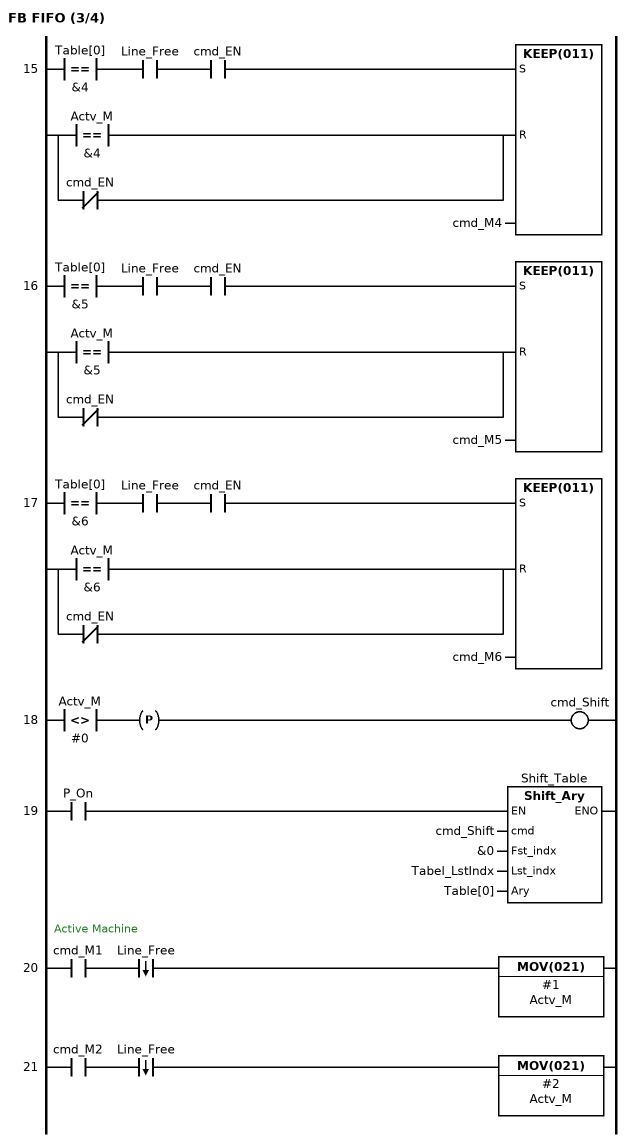
; rung 15
LD=(300) Table[0] &4
AND Line_Free
AND cmd_EN
LD=(300) Actv_M &4
ORNOT cmd_EN
KEEP(011) cmd_M4
; rung 16
LD=(300) Table[0] &5
AND Line_Free
AND cmd_EN
LD=(300) Actv_M &5
ORNOT cmd_EN
KEEP(011) cmd_M5
; rung 17
LD=(300) Table[0] &6
AND Line_Free
AND cmd_EN
LD=(300) Actv_M &6
ORNOT cmd_EN
KEEP(011) cmd_M6
; rung 18
LD<>(305) Actv_M #0
UP(521)
OUT cmd_Shift
; rung 19
LD P_On
CALL Shift_Table : Shift_Ary (cmd := cmd_Shift, Fst_indx := &0, Lst_indx := Tabel_LstIndx, Ary := Table[0])
; rung 20: Active Machine
LD cmd_M1
%AND Line_Free
MOV(021) #1 Actv_M
; rung 21
LD cmd_M2
%AND Line_Free
MOV(021) #2 Actv_M

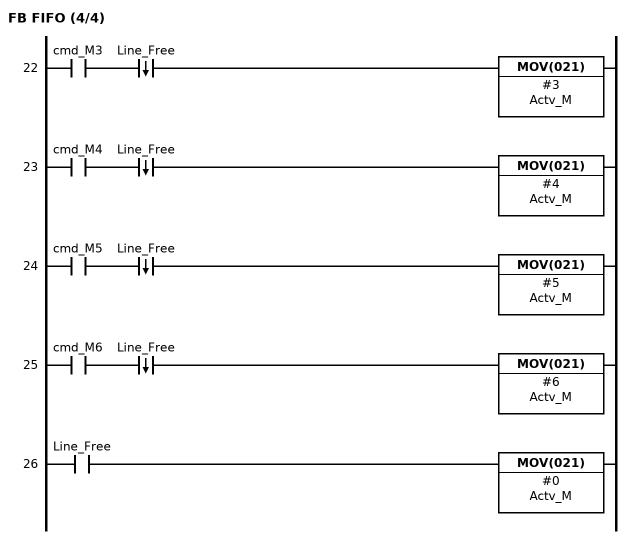
; rung 22
LD cmd_M3
%AND Line_Free
MOV(021) #3 Actv_M
; rung 23
LD cmd_M4
%AND Line_Free
MOV(021) #4 Actv_M
; rung 24
LD cmd_M5
%AND Line_Free
MOV(021) #5 Actv_M
; rung 25
LD cmd_M6
%AND Line_Free
MOV(021) #6 Actv_M
; rung 26
LD Line_Free
MOV(021) #0 Actv_M

## Function block PLC_to_MES
VAR_IN_OUT
  Dados : MqRT;
  BatchReal : s_Steps;
  Estado : s_Estado;
END_VAR
VAR
  Fnc : INT;
  P2_DInt : DINT;
  P1 : INT;
END_VAR
(* BATCH REAL *)
Fnc:= BatchReal.f;
P1:= BatchReal.p1;
P2_DInt:= REAL_TO_DINT(BatchReal.p2);

(*Limpa*)
Dados.BatchReal.Dedu.Active:= FALSE;
Dados.BatchReal.Heat.Active:= FALSE;
Dados.BatchReal.Inje.Active:= FALSE;
Dados.BatchReal.Load.Active:= FALSE;
Dados.BatchReal.Tumb.Active:= FALSE;
Dados.BatchReal.Unload.Active:= FALSE;
CASE Fnc OF 
	70: 
		Dados.BatchReal.Load.Active:= TRUE;
		Dados.BatchReal.Load.Value01:= INT_TO_DWORD(P1);
		Dados.BatchReal.Load.Value02:= DINT_TO_DWORD(P2_DInt);
	80:
		Dados.BatchReal.Unload.Active:= TRUE;
		Dados.BatchReal.Unload.Value01:= INT_TO_DWORD(P1);
		Dados.BatchReal.Unload.Value02:= DINT_TO_DWORD(P2_DInt);
	20:
		Dados.BatchReal.Heat.Active:= TRUE;
		Dados.BatchReal.Heat.Value01:= INT_TO_DWORD(P1);
		Dados.BatchReal.Heat.Value02:= DINT_TO_DWORD(P2_DInt);
	10:
		Dados.BatchReal.Dedu.Active:= TRUE;
		Dados.BatchReal.Dedu.Value01:= INT_TO_DWORD(P1);
		Dados.BatchReal.Dedu.Value02:= DINT_TO_DWORD(P2_DInt);
	40:
		Dados.BatchReal.Inje.Active:= TRUE;
		Dados.BatchReal.Inje.Value01:= INT_TO_DWORD(P1);
		Dados.BatchReal.Inje.Value02:= DINT_TO_DWORD(P2_DInt);
	30:
		Dados.BatchReal.Tumb.Active:= TRUE;
		Dados.BatchReal.Tumb.Value01:= INT_TO_DWORD(P1);
		Dados.BatchReal.Tumb.Value02:= DINT_TO_DWORD(P2_DInt);
END_CASE; 

(*ESTADOS*)
Dados.Ciclo:= Estado.Ciclo;
IF Estado.Estado AND NOT Estado.Avaria THEN
	Dados.Estado:= 1;	
ELSE
	Dados.Estado:= 0;
END_IF;
IF Estado.Manual THEN
	Dados.Estado:= 2;
END_IF;
IF Estado.FalhaInjeProd THEN
	Dados.Estado:= 3;
END_IF;
IF Estado.FalhaAquecim THEN
	Dados.Estado:= 4;
END_IF;
IF Estado.AvariaTermicos THEN
	Dados.Estado:= 5;
END_IF;
IF Estado.TratAbortado THEN
	Dados.Estado:= 6;
END_IF;
IF Estado.FalhaEnergia THEN
	Dados.Estado:= 7;
END_IF;
IF Estado.NivelProdBaixo THEN
	Dados.Estado:= 8;
END_IF;
IF Estado.Emergencia THEN
	Dados.Estado:= 9;
END_IF;
IF Dados.Estado<=2 AND Estado.Avaria THEN
	Dados.Estado:= 10;
END_IF;

IF Dados.Estado=1 THEN	
	Dados.EquiDesabil[0]:=FALSE;
ELSE
	Dados.EquiDesabil[0]:=TRUE;
END_IF;
	
Dados.FimCiclo[0]:= Estado.FimCiclo;
(*IF Estado.Avaria then
	Dados.SinAlarme:= 1;
ELSE
	Dados.SinAlarme:= 0;
END_IF;*)

## Function block RecipeCRC
VAR_INPUT
  AutoMES : BOOL;  (* Autorização MES *)
END_VAR
VAR_OUTPUT
  CRC : WORD;
END_VAR
VAR_IN_OUT
  Maq : MqDL;
END_VAR
VAR
  lenStr : INT;
  STR_Copy21 : STRING;
  STR_Copy22 : STRING;
  STR_Copy23 : STRING;
  STR_Copy24 : STRING;
  STR_Copy25 : STRING;
  STR_Copy26 : STRING;
  STR_Copy27 : STRING;
  STR_Copy28 : STRING;
  STR_Copy29 : STRING;
  STR_Copy30 : STRING;
  STR_Copy31 : STRING;
  STR_Copy32 : STRING;
  STR_Copy33 : STRING;
  STR_Copy34 : STRING;
  STR_Copy35 : STRING;
  STR_Copy36 : STRING;
  STR_Copy37 : STRING;
  STR_Copy38 : STRING;
  STR_Copy39 : STRING;
  STR_Copy40 : STRING;
  STR_Copy41 : STRING;
  STR_Copy42 : STRING;
  STR_Copy43 : STRING;
  STR_Copy44 : STRING;
  STR_Copy45 : STRING;
  STR : STRING;
  CalcCRC : CRC16;
  auxStr AT E0_32000 : STRING;
  arWord AT E0_32000 : ARRAY[0..49] OF WORD;
  ArCopy : ARRAY_COPY;
  Rec : MqDL;
  STR_Copy : STRING;
  STR_Copy2 : STRING;
  STR_Copy3 : STRING;
  STR_Copy4 : STRING;
  STR_Copy5 : STRING;
  STR_Copy6 : STRING;
  STR_Copy7 : STRING;
  STR_Copy8 : STRING;
  STR_Copy9 : STRING;
  STR_Copy10 : STRING;
  STR_Copy11 : STRING;
  STR_Copy12 : STRING;
  STR_Copy13 : STRING;
  STR_Copy14 : STRING;
  STR_Copy15 : STRING;
  STR_Copy16 : STRING;
  STR_Copy17 : STRING;
  STR_Copy18 : STRING;
  STR_Copy19 : STRING;
  STR_Copy20 : STRING;
  val : DINT;
END_VAR
Rec:= Maq;

(*Nome Ordem*)
auxStr:= '';
STR:= DINT_TO_STRING(Rec.Ordem_BL );
lenStr:= LEN(STR) ;
IF lenStr>0 THEN
	(*Autorização MES*)
	IF AutoMES THEN
		STR:= '1';
	ELSE 
		STR := '0';
	END_IF; 
	lenStr:= LEN(STR) ;
	CalcCRC(EN:= TRUE,Bytes_Qty := lenStr ,Swap:= FALSE ,CRC_Ini := 16#FFFF,Str:= STR ,CRC16=>CRC);
	STR_Copy44 := STR ;

	(*Cliente*)
	auxStr:= '';
	ArCopy (EN:= TRUE ,NPos:= 50 ,ArIN := Rec.Cliente_BL[0],ArOUT := arWord[0]);
	 STR := auxStr ;
	lenStr:= LEN(STR) ;
	IF lenStr>0 then
	CalcCRC(EN:= TRUE,Bytes_Qty := lenStr ,Swap:= FALSE ,CRC_Ini := CRC,Str:= STR ,CRC16=>CRC);
	END_IF; 
	STR_Copy := STR ;


	(*Artigo*)
	auxStr:= '';
	ArCopy (EN:= TRUE , NPos:= 50 , ArIN := Rec.Artigo_BL[0] , ArOUT := arWord[0]);
	 STR := auxStr ;
	lenStr:= LEN(STR) ;
	IF lenStr>0 then
	CalcCRC(EN:= TRUE,Bytes_Qty := lenStr ,Swap:= FALSE ,CRC_Ini := CRC,Str:= STR ,CRC16=>CRC);
	END_IF; 
	STR_Copy2 := STR ;


	(*Encomenda*)
	auxStr:= '';
	ArCopy (EN:= TRUE , NPos:= 50 , ArIN := Rec.Encomenda_BL[0] , ArOUT := arWord[0]);
	 STR := auxStr ;
	lenStr:= LEN(STR) ;
	IF lenStr>0 then
	CalcCRC(EN:= TRUE,Bytes_Qty := lenStr ,Swap:= FALSE ,CRC_Ini := CRC,Str:= STR ,CRC16=>CRC);
	END_IF; 
	STR_Copy3 := STR ;


	(*Qtd Encomenda*)
	auxStr:= '';
	STR:= UDINT_TO_STRING(Rec.QtdEncom_BL );
	lenStr:= LEN(STR) ;
	IF lenStr>0 then
	CalcCRC(EN:= TRUE,Bytes_Qty := lenStr ,Swap:= FALSE ,CRC_Ini := CRC,Str:= STR ,CRC16=>CRC);
	END_IF; 
	STR_Copy4 := STR ;


	(*Qtd Real*)
	auxStr:= '';
	STR:= UDINT_TO_STRING(Rec.QtdReal_BL );
	lenStr:= LEN(STR) ;
	IF lenStr>0 then
	CalcCRC(EN:= TRUE,Bytes_Qty := lenStr ,Swap:= FALSE ,CRC_Ini := CRC,Str:= STR ,CRC16=>CRC);
	END_IF; 
	STR_Copy5 := STR ;


	(*Data Expediçãp*)
	auxStr:= '';
	ArCopy (EN:= TRUE , NPos:= 4 , ArIN := Rec.DataExpedic_BL[0] , ArOUT := arWord[0]);
	 STR := auxStr ;
	lenStr:= LEN(STR) ;
	IF lenStr>0 then
	CalcCRC(EN:= TRUE,Bytes_Qty := lenStr ,Swap:= FALSE ,CRC_Ini := CRC,Str:= STR ,CRC16=>CRC);
	END_IF; 
	STR_Copy6 := STR ;


	(*Nome Receita*)
	auxStr:= '';
	ArCopy (EN:= TRUE , NPos:= 50 , ArIN := Rec.NomeReceita_BL[0] , ArOUT := arWord[0]);
	 STR := auxStr ;
	lenStr:= LEN(STR) ;
	IF lenStr>0 then
	CalcCRC(EN:= TRUE,Bytes_Qty := lenStr ,Swap:= FALSE ,CRC_Ini := CRC,Str:= STR ,CRC16=>CRC);
	END_IF; 
	STR_Copy7 := STR ;


	(* Ordem*)
	auxStr:= '';
	STR:= DINT_TO_STRING(Rec.Ordem_BL );
	lenStr:= LEN(STR) ;
	IF lenStr>0 then
	CalcCRC(EN:= TRUE,Bytes_Qty := lenStr ,Swap:= FALSE ,CRC_Ini := CRC,Str:= STR ,CRC16=>CRC);
	END_IF; 
	STR_Copy45 := STR ;


	(*Step Function*)
	val:= DWORD_TO_DINT(Rec.Steps_BL[0].Func ); 
	STR:= '';
	STR:= DINT_TO_STRING(val );
	lenStr:= LEN(STR) ;
	IF lenStr>0 then
	CalcCRC(EN:= TRUE,Bytes_Qty := lenStr ,Swap:= FALSE ,CRC_Ini := CRC,Str:= STR ,CRC16=>CRC);
	END_IF; 
	STR_Copy8 := STR ;

	(*Step Param01*)
	Val:= DWORD_TO_DINT(Rec.Steps_BL[0].Param01 ); 
	STR:= '';
	STR:= DINT_TO_STRING(val);
	lenStr:= LEN(STR) ;
	IF lenStr>0 then
	CalcCRC(EN:= TRUE,Bytes_Qty := lenStr ,Swap:= FALSE ,CRC_Ini := CRC,Str:= STR ,CRC16=>CRC);
	END_IF; 
	STR_Copy9 := STR ;

	(*Step Param02*)
	Val:= DWORD_TO_DINT(Rec.Steps_BL[0].Param02 ); 
	STR:= '';
	STR:= DINT_TO_STRING(val);
	lenStr:= LEN(STR) ;
	IF lenStr>0 then
	CalcCRC(EN:= TRUE,Bytes_Qty := lenStr ,Swap:= FALSE ,CRC_Ini := CRC,Str:= STR ,CRC16=>CRC);
	END_IF; 
	STR_Copy10 := STR ;


	(*Step Function*)
	val:= DWORD_TO_DINT(Rec.Steps_BL[1].Func ); 
	STR:= '';
	STR:= DINT_TO_STRING(val);
	lenStr:= LEN(STR) ;
	IF lenStr>0 then
	CalcCRC(EN:= TRUE,Bytes_Qty := lenStr ,Swap:= FALSE ,CRC_Ini := CRC,Str:= STR ,CRC16=>CRC);
	END_IF; 
	STR_Copy11 := STR ;

	(*Step Param01*)
	Val:= DWORD_TO_DINT(Rec.Steps_BL[1].Param01 ); 
	STR:= '';
	STR:= DINT_TO_STRING(val);
	lenStr:= LEN(STR) ;
	IF lenStr>0 then
	CalcCRC(EN:= TRUE,Bytes_Qty := lenStr ,Swap:= FALSE ,CRC_Ini := CRC,Str:= STR ,CRC16=>CRC);
	END_IF; 
	STR_Copy12 := STR ;

	(*Step Param02*)
	Val:= DWORD_TO_DINT(Rec.Steps_BL[1].Param02 ); 
	STR:= '';
	STR:= DINT_TO_STRING(val);
	lenStr:= LEN(STR) ;
	IF lenStr>0 then
	CalcCRC(EN:= TRUE,Bytes_Qty := lenStr ,Swap:= FALSE ,CRC_Ini := CRC,Str:= STR ,CRC16=>CRC);
	END_IF; 
	STR_Copy13 := STR ;


	(*Step Function*)
	Val:= DWORD_TO_DINT(Rec.Steps_BL[2].Func ); 
	STR:= '';
	STR:= DINT_TO_STRING(val);
	lenStr:= LEN(STR) ;
	IF lenStr>0 then
	CalcCRC(EN:= TRUE,Bytes_Qty := lenStr ,Swap:= FALSE ,CRC_Ini := CRC,Str:= STR ,CRC16=>CRC);
	END_IF; 
	STR_Copy14 := STR ;

	(*Step Param01*)
	Val:= DWORD_TO_DINT(Rec.Steps_BL[2].Param01 ); 
	STR:= '';
	STR:= DINT_TO_STRING(val);
	lenStr:= LEN(STR) ;
	IF lenStr>0 then
	CalcCRC(EN:= TRUE,Bytes_Qty := lenStr ,Swap:= FALSE ,CRC_Ini := CRC,Str:= STR ,CRC16=>CRC);
	END_IF; 
	STR_Copy15 := STR ;

	(*Step Param02*)
	Val:= DWORD_TO_DINT(Rec.Steps_BL[2].Param02 ); 
	STR:= '';
	STR:= DINT_TO_STRING(val);
	lenStr:= LEN(STR) ;
	IF lenStr>0 then
	CalcCRC(EN:= TRUE,Bytes_Qty := lenStr ,Swap:= FALSE ,CRC_Ini := CRC,Str:= STR ,CRC16=>CRC);
	END_IF; 
	STR_Copy16 := STR ;


	(*Step Function*)
	Val:= DWORD_TO_DINT(Rec.Steps_BL[3].Func ); 
	STR:= '';
	STR:= DINT_TO_STRING(val);
	lenStr:= LEN(STR) ;
	IF lenStr>0 then
	CalcCRC(EN:= TRUE,Bytes_Qty := lenStr ,Swap:= FALSE ,CRC_Ini := CRC,Str:= STR ,CRC16=>CRC);
	END_IF; 
	STR_Copy17 := STR ;

	(*Step Param01*)
	Val:= DWORD_TO_DINT(Rec.Steps_BL[3].Param01 ); 
	STR:= '';
	STR:= DINT_TO_STRING(val);
	lenStr:= LEN(STR) ;
	IF lenStr>0 then
	CalcCRC(EN:= TRUE,Bytes_Qty := lenStr ,Swap:= FALSE ,CRC_Ini := CRC,Str:= STR ,CRC16=>CRC);
	END_IF; 
	STR_Copy18 := STR ;

	(*Step Param02*)
	Val:= DWORD_TO_DINT(Rec.Steps_BL[3].Param02 ); 
	STR:= '';
	STR:= DINT_TO_STRING(val);
	lenStr:= LEN(STR) ;
	IF lenStr>0 then
	CalcCRC(EN:= TRUE,Bytes_Qty := lenStr ,Swap:= FALSE ,CRC_Ini := CRC,Str:= STR ,CRC16=>CRC);
	END_IF; 
	STR_Copy19 := STR ;


	(*Step Function*)
	Val:= DWORD_TO_DINT(Rec.Steps_BL[4].Func ); 
	STR:= '';
	STR:= DINT_TO_STRING(val);
	lenStr:= LEN(STR) ;
	IF lenStr>0 then
	CalcCRC(EN:= TRUE,Bytes_Qty := lenStr ,Swap:= FALSE ,CRC_Ini := CRC,Str:= STR ,CRC16=>CRC);
	END_IF; 
	STR_Copy20 := STR ;

	(*Step Param01*)
	Val:= DWORD_TO_DINT(Rec.Steps_BL[4].Param01 ); 
	STR:= '';
	STR:= DINT_TO_STRING(val);
	lenStr:= LEN(STR) ;
	IF lenStr>0 then
	CalcCRC(EN:= TRUE,Bytes_Qty := lenStr ,Swap:= FALSE ,CRC_Ini := CRC,Str:= STR ,CRC16=>CRC);
	END_IF; 
	STR_Copy21 := STR ;

	(*Step Param02*)
	Val:= DWORD_TO_DINT(Rec.Steps_BL[4].Param02 ); 
	STR:= '';
	STR:= DINT_TO_STRING(val);
	lenStr:= LEN(STR) ;
	IF lenStr>0 then
	CalcCRC(EN:= TRUE,Bytes_Qty := lenStr ,Swap:= FALSE ,CRC_Ini := CRC,Str:= STR ,CRC16=>CRC);
	END_IF; 
	STR_Copy22:= STR ;


	(*Step Function*)
	Val:= DWORD_TO_DINT(Rec.Steps_BL[5].Func ); 
	STR:= '';
	STR:= DINT_TO_STRING(val);
	lenStr:= LEN(STR) ;
	IF lenStr>0 then
	CalcCRC(EN:= TRUE,Bytes_Qty := lenStr ,Swap:= FALSE ,CRC_Ini := CRC,Str:= STR ,CRC16=>CRC);
	END_IF; 
	STR_Copy23 := STR ;

	(*Step Param01*)
	Val:= DWORD_TO_DINT(Rec.Steps_BL[5].Param01 ); 
	STR:= '';
	STR:= DINT_TO_STRING(val);
	lenStr:= LEN(STR) ;
	IF lenStr>0 then
	CalcCRC(EN:= TRUE,Bytes_Qty := lenStr ,Swap:= FALSE ,CRC_Ini := CRC,Str:= STR ,CRC16=>CRC);
	END_IF; 
	STR_Copy24 := STR ;

	(*Step Param02*)
	Val:= DWORD_TO_DINT(Rec.Steps_BL[5].Param02 ); 
	STR:= '';
	STR:= DINT_TO_STRING(val);
	lenStr:= LEN(STR) ;
	IF lenStr>0 then
	CalcCRC(EN:= TRUE,Bytes_Qty := lenStr ,Swap:= FALSE ,CRC_Ini := CRC,Str:= STR ,CRC16=>CRC);
	END_IF; 
	STR_Copy25 := STR ;


	(*Step Function*)
	Val:= DWORD_TO_DINT(Rec.Steps_BL[6].Func ); 
	STR:= '';
	STR:= DINT_TO_STRING(val);
	lenStr:= LEN(STR) ;
	IF lenStr>0 then
	CalcCRC(EN:= TRUE,Bytes_Qty := lenStr ,Swap:= FALSE ,CRC_Ini := CRC,Str:= STR ,CRC16=>CRC);
	END_IF; 
	STR_Copy26 := STR ;

	(*Step Param01*)
	Val:= DWORD_TO_DINT(Rec.Steps_BL[6].Param01 ); 
	STR:= '';
	STR:= DINT_TO_STRING(val);
	lenStr:= LEN(STR) ;
	IF lenStr>0 then
	CalcCRC(EN:= TRUE,Bytes_Qty := lenStr ,Swap:= FALSE ,CRC_Ini := CRC,Str:= STR ,CRC16=>CRC);
	END_IF; 
	STR_Copy27 := STR ;

	(*Step Param02*)
	Val:= DWORD_TO_DINT(Rec.Steps_BL[6].Param02 ); 
	STR:= '';
	STR:= DINT_TO_STRING(val);
	lenStr:= LEN(STR) ;
	IF lenStr>0 then
	CalcCRC(EN:= TRUE,Bytes_Qty := lenStr ,Swap:= FALSE ,CRC_Ini := CRC,Str:= STR ,CRC16=>CRC);
	END_IF; 
	STR_Copy28 := STR ;


	(*Step Function*)
	Val:= DWORD_TO_DINT(Rec.Steps_BL[7].Func ); 
	STR:= '';
	STR:= DINT_TO_STRING(val);
	lenStr:= LEN(STR) ;
	IF lenStr>0 then
	CalcCRC(EN:= TRUE,Bytes_Qty := lenStr ,Swap:= FALSE ,CRC_Ini := CRC,Str:= STR ,CRC16=>CRC);
	END_IF; 
	STR_Copy29 := STR ;

	(*Step Param01*)
	Val:= DWORD_TO_DINT(Rec.Steps_BL[7].Param01 ); 
	STR:= '';
	STR:= DINT_TO_STRING(val);
	lenStr:= LEN(STR) ;
	IF lenStr>0 then
	CalcCRC(EN:= TRUE,Bytes_Qty := lenStr ,Swap:= FALSE ,CRC_Ini := CRC,Str:= STR ,CRC16=>CRC);
	END_IF; 
	STR_Copy30 := STR ;

	(*Step Param02*)
	Val:= DWORD_TO_DINT(Rec.Steps_BL[7].Param02 ); 
	STR:= '';
	STR:= DINT_TO_STRING(val);
	lenStr:= LEN(STR) ;
	IF lenStr>0 then
	CalcCRC(EN:= TRUE,Bytes_Qty := lenStr ,Swap:= FALSE ,CRC_Ini := CRC,Str:= STR ,CRC16=>CRC);
	END_IF; 
	STR_Copy31 := STR ;


	(*Step Function*)
	Val:= DWORD_TO_DINT(Rec.Steps_BL[8].Func ); 
	STR:= '';
	STR:= DINT_TO_STRING(val);
	lenStr:= LEN(STR) ;
	IF lenStr>0 then
	CalcCRC(EN:= TRUE,Bytes_Qty := lenStr ,Swap:= FALSE ,CRC_Ini := CRC,Str:= STR ,CRC16=>CRC);
	END_IF; 
	STR_Copy32 := STR ;

	(*Step Param01*)
	Val:= DWORD_TO_DINT(Rec.Steps_BL[8].Param01 ); 
	STR:= '';
	STR:= DINT_TO_STRING(val);
	lenStr:= LEN(STR) ;
	IF lenStr>0 then
	CalcCRC(EN:= TRUE,Bytes_Qty := lenStr ,Swap:= FALSE ,CRC_Ini := CRC,Str:= STR ,CRC16=>CRC);
	END_IF; 
	STR_Copy33 := STR ;

	(*Step Param02*)
	Val:= DWORD_TO_DINT(Rec.Steps_BL[8].Param02 ); 
	STR:= '';
	STR:= DINT_TO_STRING(val);
	lenStr:= LEN(STR) ;
	IF lenStr>0 then
	CalcCRC(EN:= TRUE,Bytes_Qty := lenStr ,Swap:= FALSE ,CRC_Ini := CRC,Str:= STR ,CRC16=>CRC);
	END_IF; 
	STR_Copy34 := STR ;


	(*Step Function*)
	Val:= DWORD_TO_DINT(Rec.Steps_BL[9].Func ); 
	STR:= '';
	STR:= DINT_TO_STRING(val);
	lenStr:= LEN(STR) ;
	IF lenStr>0 then
	CalcCRC(EN:= TRUE,Bytes_Qty := lenStr ,Swap:= FALSE ,CRC_Ini := CRC,Str:= STR ,CRC16=>CRC);
	END_IF; 
	STR_Copy35 := STR ;

	(*Step Param01*)
	Val:= DWORD_TO_DINT(Rec.Steps_BL[9].Param01 ); 
	STR:= '';
	STR:= DINT_TO_STRING(val);
	lenStr:= LEN(STR) ;
	IF lenStr>0 then
	CalcCRC(EN:= TRUE,Bytes_Qty := lenStr ,Swap:= FALSE ,CRC_Ini := CRC,Str:= STR ,CRC16=>CRC);
	END_IF; 
	STR_Copy36 := STR ;

	(*Step Param02*)
	Val:= DWORD_TO_DINT(Rec.Steps_BL[9].Param02 ); 
	STR:= '';
	STR:= DINT_TO_STRING(val);
	lenStr:= LEN(STR) ;
	IF lenStr>0 then
	CalcCRC(EN:= TRUE,Bytes_Qty := lenStr ,Swap:= FALSE ,CRC_Ini := CRC,Str:= STR ,CRC16=>CRC);
	END_IF; 
	STR_Copy37 := STR ;


	(*Step Function*)
	Val:= DWORD_TO_DINT(Rec.Steps_BL[10].Func ); 
	STR:= '';
	STR:= DINT_TO_STRING(val);
	lenStr:= LEN(STR) ;
	IF lenStr>0 then
	CalcCRC(EN:= TRUE,Bytes_Qty := lenStr ,Swap:= FALSE ,CRC_Ini := CRC,Str:= STR ,CRC16=>CRC);
	END_IF; 
	STR_Copy38 := STR ;

	(*Step Param01*)
	Val:= DWORD_TO_DINT(Rec.Steps_BL[10].Param01 ); 
	STR:= '';
	STR:= DINT_TO_STRING(val);
	lenStr:= LEN(STR) ;
	IF lenStr>0 then
	CalcCRC(EN:= TRUE,Bytes_Qty := lenStr ,Swap:= FALSE ,CRC_Ini := CRC,Str:= STR ,CRC16=>CRC);
	END_IF; 
	STR_Copy39 := STR ;

	(*Step Param02*)
	Val:= DWORD_TO_DINT(Rec.Steps_BL[10].Param02 ); 
	STR:= '';
	STR:= DINT_TO_STRING(val);
	lenStr:= LEN(STR) ;
	IF lenStr>0 then
	CalcCRC(EN:= TRUE,Bytes_Qty := lenStr ,Swap:= FALSE ,CRC_Ini := CRC,Str:= STR ,CRC16=>CRC);
	END_IF; 
	STR_Copy40 := STR ;


	(*Step Function*)
	Val:= DWORD_TO_DINT(Rec.Steps_BL[11].Func ); 
	STR:= '';
	STR:= DINT_TO_STRING(val);
	lenStr:= LEN(STR) ;
	IF lenStr>0 then
	CalcCRC(EN:= TRUE,Bytes_Qty := lenStr ,Swap:= FALSE ,CRC_Ini := CRC,Str:= STR ,CRC16=>CRC);
	END_IF; 
	STR_Copy41 := STR ;

	(*Step Param01*)
	Val:= DWORD_TO_DINT(Rec.Steps_BL[11].Param01 ); 
	STR:= '';
	STR:= DINT_TO_STRING(val);
	lenStr:= LEN(STR) ;
	IF lenStr>0 then
	CalcCRC(EN:= TRUE,Bytes_Qty := lenStr ,Swap:= FALSE ,CRC_Ini := CRC,Str:= STR ,CRC16=>CRC);
	END_IF; 
	STR_Copy42 := STR ;

	(*Step Param02*)
	Val:= DWORD_TO_DINT(Rec.Steps_BL[11].Param02 ); 
	STR:= '';
	STR:= DINT_TO_STRING(val);
	lenStr:= LEN(STR) ;
	IF lenStr>0 then
	CalcCRC(EN:= TRUE,Bytes_Qty := lenStr ,Swap:= FALSE ,CRC_Ini := CRC,Str:= STR ,CRC16=>CRC);
	END_IF; 
	STR_Copy43 := STR ;
ELSE
	CRC:= 0;
END_IF;

## Function block RecipeTranslate
VAR_IN_OUT
  Dados : MqDL;
  Receita : s_of;
END_VAR
VAR
  P2_DInt : DINT;
END_VAR
Receita.cliente.DataExpedicao[0]:= Dados.DataExpedic_BL[0];
Receita.cliente.DataExpedicao[1]:= Dados.DataExpedic_BL[1];
Receita.cliente.DataExpedicao[2]:= Dados.DataExpedic_BL[2];
Receita.cliente.DataExpedicao[3]:= Dados.DataExpedic_BL[3];
Receita.cliente.QtdEncomenda:= Dados.QtdEncom_BL;
Receita.cliente.QtdReal:= Dados.QtdReal_BL;

(* 0 *)
(*Step Function*)
Receita.prg.pss[0].f:= DWORD_TO_INT(Dados.Steps_BL[0].Func);

(*Step Param01*)
Receita.prg.pss[0].p1:=DWORD_TO_INT(Dados.Steps_BL[0].Param01);

(*Step Param02*)
P2_DInt:= DWORD_TO_DINT(Dados.Steps_BL[0].Param02);
Receita.prg.pss[0].p2:=DINT_TO_REAL(P2_DInt);

(* 1 *)
(*Step Function*)
Receita.prg.pss[1].f:= DWORD_TO_INT(Dados.Steps_BL[1].Func);

(*Step Param01*)
Receita.prg.pss[1].p1:=DWORD_TO_INT(Dados.Steps_BL[1].Param01);

(*Step Param02*)
P2_DInt:= DWORD_TO_DINT(Dados.Steps_BL[1].Param02);
Receita.prg.pss[1].p2:=DINT_TO_REAL(P2_DInt);

(* 2 *)
(*Step Function*)
Receita.prg.pss[2].f:= DWORD_TO_INT(Dados.Steps_BL[2].Func);

(*Step Param01*)
Receita.prg.pss[2].p1:=DWORD_TO_INT(Dados.Steps_BL[2].Param01);

(*Step Param02*)
P2_DInt:= DWORD_TO_DINT(Dados.Steps_BL[2].Param02);
Receita.prg.pss[2].p2:=DINT_TO_REAL(P2_DInt);

(* 3 *)
(*Step Function*)
Receita.prg.pss[3].f:= DWORD_TO_INT(Dados.Steps_BL[3].Func);

(*Step Param01*)
Receita.prg.pss[3].p1:=DWORD_TO_INT(Dados.Steps_BL[3].Param01);

(*Step Param02*)
P2_DInt:= DWORD_TO_DINT(Dados.Steps_BL[3].Param02);
Receita.prg.pss[3].p2:=DINT_TO_REAL(P2_DInt);

(* 4 *)
(*Step Function*)
Receita.prg.pss[4].f:= DWORD_TO_INT(Dados.Steps_BL[4].Func);

(*Step Param01*)
Receita.prg.pss[4].p1:=DWORD_TO_INT(Dados.Steps_BL[4].Param01);

(*Step Param02*)
P2_DInt:= DWORD_TO_DINT(Dados.Steps_BL[4].Param02);
Receita.prg.pss[4].p2:=DINT_TO_REAL(P2_DInt);

(* 5 *)
(*Step Function*)
Receita.prg.pss[5].f:= DWORD_TO_INT(Dados.Steps_BL[5].Func);

(*Step Param01*)
Receita.prg.pss[5].p1:=DWORD_TO_INT(Dados.Steps_BL[5].Param01);

(*Step Param02*)
P2_DInt:= DWORD_TO_DINT(Dados.Steps_BL[5].Param02);
Receita.prg.pss[5].p2:=DINT_TO_REAL(P2_DInt);

(* 6 *)
(*Step Function*)
Receita.prg.pss[6].f:= DWORD_TO_INT(Dados.Steps_BL[6].Func);

(*Step Param01*)
Receita.prg.pss[6].p1:=DWORD_TO_INT(Dados.Steps_BL[6].Param01);

(*Step Param02*)
P2_DInt:= DWORD_TO_DINT(Dados.Steps_BL[6].Param02);
Receita.prg.pss[6].p2:=DINT_TO_REAL(P2_DInt);

(* 7 *)
(*Step Function*)
Receita.prg.pss[7].f:= DWORD_TO_INT(Dados.Steps_BL[7].Func);

(*Step Param01*)
Receita.prg.pss[7].p1:=DWORD_TO_INT(Dados.Steps_BL[7].Param01);

(*Step Param02*)
P2_DInt:= DWORD_TO_DINT(Dados.Steps_BL[7].Param02);
Receita.prg.pss[7].p2:=DINT_TO_REAL(P2_DInt);

(* 8 *)
(*Step Function*)
Receita.prg.pss[8].f:= DWORD_TO_INT(Dados.Steps_BL[8].Func);

(*Step Param01*)
Receita.prg.pss[8].p1:=DWORD_TO_INT(Dados.Steps_BL[8].Param01);

(*Step Param02*)
P2_DInt:= DWORD_TO_DINT(Dados.Steps_BL[8].Param02);
Receita.prg.pss[8].p2:=DINT_TO_REAL(P2_DInt);

(* 9 *)
(*Step Function*)
Receita.prg.pss[9].f:= DWORD_TO_INT(Dados.Steps_BL[9].Func);

(*Step Param01*)
Receita.prg.pss[9].p1:=DWORD_TO_INT(Dados.Steps_BL[9].Param01);

(*Step Param02*)
P2_DInt:= DWORD_TO_DINT(Dados.Steps_BL[9].Param02);
Receita.prg.pss[9].p2:=DINT_TO_REAL(P2_DInt);

(* 10 *)
(*Step Function*)
Receita.prg.pss[10].f:= DWORD_TO_INT(Dados.Steps_BL[10].Func);

(*Step Param01*)
Receita.prg.pss[10].p1:=DWORD_TO_INT(Dados.Steps_BL[10].Param01);

(*Step Param02*)
P2_DInt:= DWORD_TO_DINT(Dados.Steps_BL[10].Param02);
Receita.prg.pss[10].p2:=DINT_TO_REAL(P2_DInt);

(* 11 *)
(*Step Function*)
Receita.prg.pss[11].f:= DWORD_TO_INT(Dados.Steps_BL[11].Func);

(*Step Param01*)
Receita.prg.pss[11].p1:=DWORD_TO_INT(Dados.Steps_BL[11].Param01);

(*Step Param02*)
P2_DInt:= DWORD_TO_DINT(Dados.Steps_BL[11].Param02);
Receita.prg.pss[11].p2:=DINT_TO_REAL(P2_DInt);


Receita.cliente.Artigo[0]:= Dados.Artigo_BL[0];
Receita.cliente.Artigo[1]:= Dados.Artigo_BL[1];
Receita.cliente.Artigo[2]:= Dados.Artigo_BL[2];
Receita.cliente.Artigo[3]:= Dados.Artigo_BL[3];
Receita.cliente.Artigo[4]:= Dados.Artigo_BL[4];
Receita.cliente.Artigo[5]:= Dados.Artigo_BL[5];
Receita.cliente.Artigo[6]:= Dados.Artigo_BL[6];
Receita.cliente.Artigo[7]:= Dados.Artigo_BL[7];
Receita.cliente.Artigo[8]:= Dados.Artigo_BL[8];
Receita.cliente.Artigo[9]:= Dados.Artigo_BL[9];
Receita.cliente.Artigo[10]:= Dados.Artigo_BL[10];
Receita.cliente.Artigo[11]:= Dados.Artigo_BL[11];
Receita.cliente.Artigo[12]:= Dados.Artigo_BL[12];
Receita.cliente.Artigo[13]:= Dados.Artigo_BL[13];
Receita.cliente.Artigo[14]:= Dados.Artigo_BL[14];
Receita.cliente.Artigo[15]:= Dados.Artigo_BL[15];
Receita.cliente.Artigo[16]:= Dados.Artigo_BL[16];
Receita.cliente.Artigo[17]:= Dados.Artigo_BL[17];
Receita.cliente.Artigo[18]:= Dados.Artigo_BL[18];
Receita.cliente.Artigo[19]:= Dados.Artigo_BL[19];
Receita.cliente.Artigo[20]:= Dados.Artigo_BL[20];
Receita.cliente.Artigo[21]:= Dados.Artigo_BL[21];
Receita.cliente.Artigo[22]:= Dados.Artigo_BL[22];
Receita.cliente.Artigo[23]:= Dados.Artigo_BL[23];
Receita.cliente.Artigo[24]:= Dados.Artigo_BL[24];
Receita.cliente.Artigo[25]:= Dados.Artigo_BL[25];
Receita.cliente.Artigo[26]:= Dados.Artigo_BL[26];
Receita.cliente.Artigo[27]:= Dados.Artigo_BL[27];
Receita.cliente.Artigo[28]:= Dados.Artigo_BL[28];
Receita.cliente.Artigo[29]:= Dados.Artigo_BL[29];
Receita.cliente.Artigo[30]:= Dados.Artigo_BL[30];
Receita.cliente.Artigo[31]:= Dados.Artigo_BL[31];
Receita.cliente.Artigo[32]:= Dados.Artigo_BL[32];
Receita.cliente.Artigo[33]:= Dados.Artigo_BL[33];
Receita.cliente.Artigo[34]:= Dados.Artigo_BL[34];
Receita.cliente.Artigo[35]:= Dados.Artigo_BL[35];
Receita.cliente.Artigo[36]:= Dados.Artigo_BL[36];
Receita.cliente.Artigo[37]:= Dados.Artigo_BL[37];
Receita.cliente.Artigo[38]:= Dados.Artigo_BL[38];
Receita.cliente.Artigo[39]:= Dados.Artigo_BL[39];
Receita.cliente.Artigo[40]:= Dados.Artigo_BL[40];
Receita.cliente.Artigo[41]:= Dados.Artigo_BL[41];
Receita.cliente.Artigo[42]:= Dados.Artigo_BL[42];
Receita.cliente.Artigo[43]:= Dados.Artigo_BL[43];
Receita.cliente.Artigo[44]:= Dados.Artigo_BL[44];
Receita.cliente.Artigo[45]:= Dados.Artigo_BL[45];
Receita.cliente.Artigo[46]:= Dados.Artigo_BL[46];
Receita.cliente.Artigo[47]:= Dados.Artigo_BL[47];
Receita.cliente.Artigo[48]:= Dados.Artigo_BL[48];
Receita.cliente.Artigo[49]:= Dados.Artigo_BL[49];

Receita.cliente.Cliente[0]:= Dados.Cliente_BL[0];
Receita.cliente.Cliente[1]:= Dados.Cliente_BL[1];
Receita.cliente.Cliente[2]:= Dados.Cliente_BL[2];
Receita.cliente.Cliente[3]:= Dados.Cliente_BL[3];
Receita.cliente.Cliente[4]:= Dados.Cliente_BL[4];
Receita.cliente.Cliente[5]:= Dados.Cliente_BL[5];
Receita.cliente.Cliente[6]:= Dados.Cliente_BL[6];
Receita.cliente.Cliente[7]:= Dados.Cliente_BL[7];
Receita.cliente.Cliente[8]:= Dados.Cliente_BL[8];
Receita.cliente.Cliente[9]:= Dados.Cliente_BL[9];
Receita.cliente.Cliente[10]:= Dados.Cliente_BL[10];
Receita.cliente.Cliente[11]:= Dados.Cliente_BL[11];
Receita.cliente.Cliente[12]:= Dados.Cliente_BL[12];
Receita.cliente.Cliente[13]:= Dados.Cliente_BL[13];
Receita.cliente.Cliente[14]:= Dados.Cliente_BL[14];
Receita.cliente.Cliente[15]:= Dados.Cliente_BL[15];
Receita.cliente.Cliente[16]:= Dados.Cliente_BL[16];
Receita.cliente.Cliente[17]:= Dados.Cliente_BL[17];
Receita.cliente.Cliente[18]:= Dados.Cliente_BL[18];
Receita.cliente.Cliente[19]:= Dados.Cliente_BL[19];
Receita.cliente.Cliente[20]:= Dados.Cliente_BL[20];
Receita.cliente.Cliente[21]:= Dados.Cliente_BL[21];
Receita.cliente.Cliente[22]:= Dados.Cliente_BL[22];
Receita.cliente.Cliente[23]:= Dados.Cliente_BL[23];
Receita.cliente.Cliente[24]:= Dados.Cliente_BL[24];
Receita.cliente.Cliente[25]:= Dados.Cliente_BL[25];
Receita.cliente.Cliente[26]:= Dados.Cliente_BL[26];
Receita.cliente.Cliente[27]:= Dados.Cliente_BL[27];
Receita.cliente.Cliente[28]:= Dados.Cliente_BL[28];
Receita.cliente.Cliente[29]:= Dados.Cliente_BL[29];
Receita.cliente.Cliente[30]:= Dados.Cliente_BL[30];
Receita.cliente.Cliente[31]:= Dados.Cliente_BL[31];
Receita.cliente.Cliente[32]:= Dados.Cliente_BL[32];
Receita.cliente.Cliente[33]:= Dados.Cliente_BL[33];
Receita.cliente.Cliente[34]:= Dados.Cliente_BL[34];
Receita.cliente.Cliente[35]:= Dados.Cliente_BL[35];
Receita.cliente.Cliente[36]:= Dados.Cliente_BL[36];
Receita.cliente.Cliente[37]:= Dados.Cliente_BL[37];
Receita.cliente.Cliente[38]:= Dados.Cliente_BL[38];
Receita.cliente.Cliente[39]:= Dados.Cliente_BL[39];
Receita.cliente.Cliente[40]:= Dados.Cliente_BL[40];
Receita.cliente.Cliente[41]:= Dados.Cliente_BL[41];
Receita.cliente.Cliente[42]:= Dados.Cliente_BL[42];
Receita.cliente.Cliente[43]:= Dados.Cliente_BL[43];
Receita.cliente.Cliente[44]:= Dados.Cliente_BL[44];
Receita.cliente.Cliente[45]:= Dados.Cliente_BL[45];
Receita.cliente.Cliente[46]:= Dados.Cliente_BL[46];
Receita.cliente.Cliente[47]:= Dados.Cliente_BL[47];
Receita.cliente.Cliente[48]:= Dados.Cliente_BL[48];
Receita.cliente.Cliente[49]:= Dados.Cliente_BL[49];

Receita.cliente.Encomenda[0]:= Dados.Encomenda_BL[0];
Receita.cliente.Encomenda[1]:= Dados.Encomenda_BL[1];
Receita.cliente.Encomenda[2]:= Dados.Encomenda_BL[2];
Receita.cliente.Encomenda[3]:= Dados.Encomenda_BL[3];
Receita.cliente.Encomenda[4]:= Dados.Encomenda_BL[4];
Receita.cliente.Encomenda[5]:= Dados.Encomenda_BL[5];
Receita.cliente.Encomenda[6]:= Dados.Encomenda_BL[6];
Receita.cliente.Encomenda[7]:= Dados.Encomenda_BL[7];
Receita.cliente.Encomenda[8]:= Dados.Encomenda_BL[8];
Receita.cliente.Encomenda[9]:= Dados.Encomenda_BL[9];
Receita.cliente.Encomenda[10]:= Dados.Encomenda_BL[10];
Receita.cliente.Encomenda[11]:= Dados.Encomenda_BL[11];
Receita.cliente.Encomenda[12]:= Dados.Encomenda_BL[12];
Receita.cliente.Encomenda[13]:= Dados.Encomenda_BL[13];
Receita.cliente.Encomenda[14]:= Dados.Encomenda_BL[14];
Receita.cliente.Encomenda[15]:= Dados.Encomenda_BL[15];
Receita.cliente.Encomenda[16]:= Dados.Encomenda_BL[16];
Receita.cliente.Encomenda[17]:= Dados.Encomenda_BL[17];
Receita.cliente.Encomenda[18]:= Dados.Encomenda_BL[18];
Receita.cliente.Encomenda[19]:= Dados.Encomenda_BL[19];
Receita.cliente.Encomenda[20]:= Dados.Encomenda_BL[20];
Receita.cliente.Encomenda[21]:= Dados.Encomenda_BL[21];
Receita.cliente.Encomenda[22]:= Dados.Encomenda_BL[22];
Receita.cliente.Encomenda[23]:= Dados.Encomenda_BL[23];
Receita.cliente.Encomenda[24]:= Dados.Encomenda_BL[24];
Receita.cliente.Encomenda[25]:= Dados.Encomenda_BL[25];
Receita.cliente.Encomenda[26]:= Dados.Encomenda_BL[26];
Receita.cliente.Encomenda[27]:= Dados.Encomenda_BL[27];
Receita.cliente.Encomenda[28]:= Dados.Encomenda_BL[28];
Receita.cliente.Encomenda[29]:= Dados.Encomenda_BL[29];
Receita.cliente.Encomenda[30]:= Dados.Encomenda_BL[30];
Receita.cliente.Encomenda[31]:= Dados.Encomenda_BL[31];
Receita.cliente.Encomenda[32]:= Dados.Encomenda_BL[32];
Receita.cliente.Encomenda[33]:= Dados.Encomenda_BL[33];
Receita.cliente.Encomenda[34]:= Dados.Encomenda_BL[34];
Receita.cliente.Encomenda[35]:= Dados.Encomenda_BL[35];
Receita.cliente.Encomenda[36]:= Dados.Encomenda_BL[36];
Receita.cliente.Encomenda[37]:= Dados.Encomenda_BL[37];
Receita.cliente.Encomenda[38]:= Dados.Encomenda_BL[38];
Receita.cliente.Encomenda[39]:= Dados.Encomenda_BL[39];
Receita.cliente.Encomenda[40]:= Dados.Encomenda_BL[40];
Receita.cliente.Encomenda[41]:= Dados.Encomenda_BL[41];
Receita.cliente.Encomenda[42]:= Dados.Encomenda_BL[42];
Receita.cliente.Encomenda[43]:= Dados.Encomenda_BL[43];
Receita.cliente.Encomenda[44]:= Dados.Encomenda_BL[44];
Receita.cliente.Encomenda[45]:= Dados.Encomenda_BL[45];
Receita.cliente.Encomenda[46]:= Dados.Encomenda_BL[46];
Receita.cliente.Encomenda[47]:= Dados.Encomenda_BL[47];
Receita.cliente.Encomenda[48]:= Dados.Encomenda_BL[48];
Receita.cliente.Encomenda[49]:= Dados.Encomenda_BL[49];

Receita.cliente.NomeReceita[0]:= Dados.NomeReceita_BL[0];
Receita.cliente.NomeReceita[1]:= Dados.NomeReceita_BL[1];
Receita.cliente.NomeReceita[2]:= Dados.NomeReceita_BL[2];
Receita.cliente.NomeReceita[3]:= Dados.NomeReceita_BL[3];
Receita.cliente.NomeReceita[4]:= Dados.NomeReceita_BL[4];
Receita.cliente.NomeReceita[5]:= Dados.NomeReceita_BL[5];
Receita.cliente.NomeReceita[6]:= Dados.NomeReceita_BL[6];
Receita.cliente.NomeReceita[7]:= Dados.NomeReceita_BL[7];
Receita.cliente.NomeReceita[8]:= Dados.NomeReceita_BL[8];
Receita.cliente.NomeReceita[9]:= Dados.NomeReceita_BL[9];
Receita.cliente.NomeReceita[10]:= Dados.NomeReceita_BL[10];
Receita.cliente.NomeReceita[11]:= Dados.NomeReceita_BL[11];
Receita.cliente.NomeReceita[12]:= Dados.NomeReceita_BL[12];
Receita.cliente.NomeReceita[13]:= Dados.NomeReceita_BL[13];
Receita.cliente.NomeReceita[14]:= Dados.NomeReceita_BL[14];
Receita.cliente.NomeReceita[15]:= Dados.NomeReceita_BL[15];
Receita.cliente.NomeReceita[16]:= Dados.NomeReceita_BL[16];
Receita.cliente.NomeReceita[17]:= Dados.NomeReceita_BL[17];
Receita.cliente.NomeReceita[18]:= Dados.NomeReceita_BL[18];
Receita.cliente.NomeReceita[19]:= Dados.NomeReceita_BL[19];
Receita.cliente.NomeReceita[20]:= Dados.NomeReceita_BL[20];
Receita.cliente.NomeReceita[21]:= Dados.NomeReceita_BL[21];
Receita.cliente.NomeReceita[22]:= Dados.NomeReceita_BL[22];
Receita.cliente.NomeReceita[23]:= Dados.NomeReceita_BL[23];
Receita.cliente.NomeReceita[24]:= Dados.NomeReceita_BL[24];
Receita.cliente.NomeReceita[25]:= Dados.NomeReceita_BL[25];
Receita.cliente.NomeReceita[26]:= Dados.NomeReceita_BL[26];
Receita.cliente.NomeReceita[27]:= Dados.NomeReceita_BL[27];
Receita.cliente.NomeReceita[28]:= Dados.NomeReceita_BL[28];
Receita.cliente.NomeReceita[29]:= Dados.NomeReceita_BL[29];
Receita.cliente.NomeReceita[30]:= Dados.NomeReceita_BL[30];
Receita.cliente.NomeReceita[31]:= Dados.NomeReceita_BL[31];
Receita.cliente.NomeReceita[32]:= Dados.NomeReceita_BL[32];
Receita.cliente.NomeReceita[33]:= Dados.NomeReceita_BL[33];
Receita.cliente.NomeReceita[34]:= Dados.NomeReceita_BL[34];
Receita.cliente.NomeReceita[35]:= Dados.NomeReceita_BL[35];
Receita.cliente.NomeReceita[36]:= Dados.NomeReceita_BL[36];
Receita.cliente.NomeReceita[37]:= Dados.NomeReceita_BL[37];
Receita.cliente.NomeReceita[38]:= Dados.NomeReceita_BL[38];
Receita.cliente.NomeReceita[39]:= Dados.NomeReceita_BL[39];
Receita.cliente.NomeReceita[40]:= Dados.NomeReceita_BL[40];
Receita.cliente.NomeReceita[41]:= Dados.NomeReceita_BL[41];
Receita.cliente.NomeReceita[42]:= Dados.NomeReceita_BL[42];
Receita.cliente.NomeReceita[43]:= Dados.NomeReceita_BL[43];
Receita.cliente.NomeReceita[44]:= Dados.NomeReceita_BL[44];
Receita.cliente.NomeReceita[45]:= Dados.NomeReceita_BL[45];
Receita.cliente.NomeReceita[46]:= Dados.NomeReceita_BL[46];
Receita.cliente.NomeReceita[47]:= Dados.NomeReceita_BL[47];
Receita.cliente.NomeReceita[48]:= Dados.NomeReceita_BL[48];
Receita.cliente.NomeReceita[49]:= Dados.NomeReceita_BL[49];

## Function block RecipeTst
VAR_INPUT
  Star : BOOL;
  AreaID : INT;
  IniSteps : UDINT;
  NSteps : INT;  (* Nº passos da receita *)
END_VAR
VAR_OUTPUT
  Recipe_Ok : BOOL;
END_VAR
VAR_IN_OUT
  Recipe_NOK : ARRAY[0..15] OF BOOL;
END_VAR
VAR
  Function : DWORD;
  Param01 : DWORD;
  Param02 : DWORD;
  i : UINT;
  typeDM AT D0 : WORD;
  typeEM AT E0_0 : WORD;
  aux : ARRAY[0..1] OF WORD;
  bit_NOK : BOOL;
  Par1 : DWORD;
  Par2 : DWORD;
  bit_Par1_Ok : BOOL;
  bit_Par2_Ok : BOOL;
  converter : DWord_To_Real;
  valor : REAL;
END_VAR

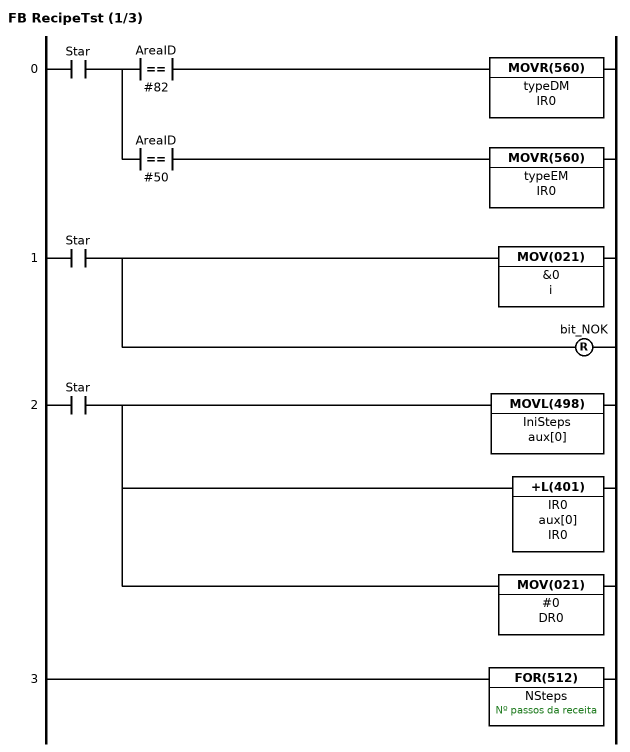
; rung 0
LD Star
OUT TR0
AND=(300) AreaID #82
MOVR(560) typeDM IR0
LD TR0
AND=(300) AreaID #50
MOVR(560) typeEM IR0
; rung 1
LD Star
MOV(021) &0 i
RSET bit_NOK
; rung 2
LD Star
MOVL(498) IniSteps aux[0]
+L(401) IR0 aux[0] IR0
MOV(021) #0 DR0
; rung 3
FOR(512) NSteps  ; Nº passos da receita

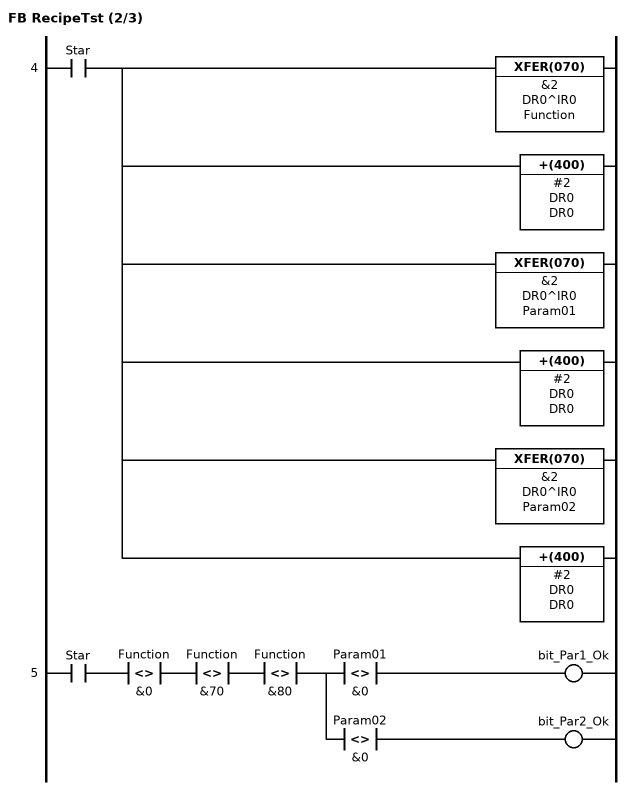
; rung 4
LD Star
XFER(070) &2 DR0^IR0 Function
+(400) #2 DR0 DR0
XFER(070) &2 DR0^IR0 Param01
+(400) #2 DR0 DR0
XFER(070) &2 DR0^IR0 Param02
+(400) #2 DR0 DR0
; rung 5
LD Star
AND<>(305) Function &0
AND<>(305) Function &70
AND<>(305) Function &80
OUT TR0
AND<>(305) Param01 &0
OUT bit_Par1_Ok
LD TR0
AND<>(305) Param02 &0
OUT bit_Par2_Ok

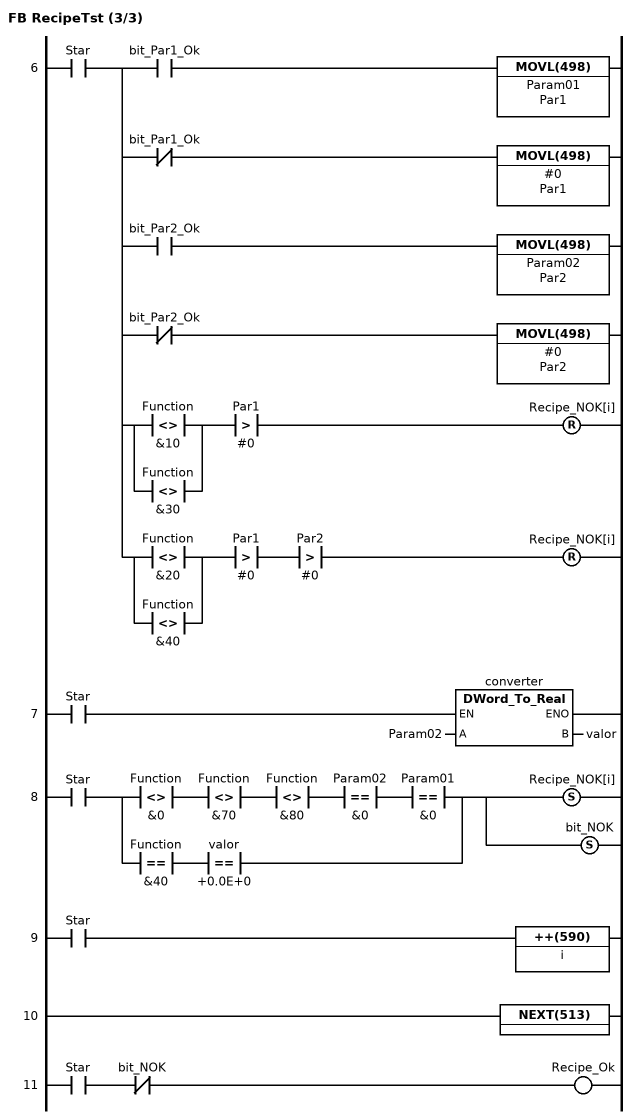
; rung 6
LD Star
OUT TR0
AND bit_Par1_Ok
MOVL(498) Param01 Par1
LD TR0
ANDNOT bit_Par1_Ok
MOVL(498) #0 Par1
LD TR0
AND bit_Par2_Ok
MOVL(498) Param02 Par2
LD TR0
ANDNOT bit_Par2_Ok
MOVL(498) #0 Par2
LD TR0
LD<>(305) Function &10
OR<>(305) Function &30
ANDLD
AND>(320) Par1 #0
RSET Recipe_NOK[i]
LD TR0
LD<>(305) Function &20
OR<>(305) Function &40
ANDLD
AND>(320) Par1 #0
AND>(320) Par2 #0
RSET Recipe_NOK[i]
; rung 7
LD Star
CALL converter : DWord_To_Real (A := Param02, B => valor)
; rung 8
LD Star
LD<>(305) Function &0
AND<>(305) Function &70
AND<>(305) Function &80
AND=(300) Param02 &0
AND=(300) Param01 &0
LD=(300) Function &40
AND=F(329) valor +0.0E+0
ORLD
ANDLD
SET Recipe_NOK[i]
SET bit_NOK
; rung 9
LD Star
++(590) i
; rung 10
NEXT(513)
; rung 11
LD Star
ANDNOT bit_NOK
OUT Recipe_Ok

## Function block Shift_Ary
VAR_INPUT
  cmd : BOOL;
  Fst_indx : INT;
  Lst_indx : INT;
END_VAR
VAR_IN_OUT
  Ary : ARRAY[0..99] OF INT;
END_VAR
VAR
  itr : INT;
  nxt_itr : INT;
END_VAR
IF cmd THEN
	
FOR itr := Fst_indx TO Lst_indx-1 DO
	nxt_itr := itr+1;
Ary[itr] := Ary[nxt_itr];
END_FOR;

Ary[Lst_indx] := 0;

END_IF;

## Function block Str_To_Real
VAR_OUTPUT
  Valor : REAL;
END_VAR
VAR_IN_OUT
  Str : STRING;
END_VAR
VAR
  auxDInt : DINT;
END_VAR
auxDInt:= STRING_TO_DINT (Str);
Valor:=DINT_TO_REAL(auxDInt);